LIN {X 0,Y 641.968,Z 762.06,A -85,B 0,C 180,E1 5618.929,E2 5618.929} C_VEL
LIN {X 0,Y 642.524,Z 763.494,A -85,B 0,C 180,E1 5625.268,E2 5625.268} C_VEL
LIN {X 0,Y 669.251,Z 813.676,A -85,B 0,C 180,E1 5628.22,E2 5628.22} C_VEL
LIN {X 0,Y 666.394,Z 892.129,A -85,B 0,C 180,E1 5629.884,E2 5629.884} C_VEL
LIN {X 0,Y 661.27,Z 964.972,A -85,B 0,C 180,E1 5632.787,E2 5632.787} C_VEL
LIN {X 0,Y 655.013,Z 1034.337,A -85,B 0,C 180,E1 5637.06,E2 5637.06} C_VEL
LIN {X 0,Y 649.321,Z 1095.62,A -85,B 0,C 180,E1 5642.548,E2 5642.548} C_VEL
LIN {X 0,Y 645.565,Z 1141.854,A -85,B 0,C 180,E1 5648.388,E2 5648.388} C_VEL
LIN {X 0,Y 643.703,Z 1174.825,A -85,B 0,C 180,E1 5654.309,E2 5654.309} C_VEL
LIN {X 0,Y 643.008,Z 1195.415,A -85,B 0,C 180,E1 5659.842,E2 5659.842} C_VEL
LIN {X 0,Y 642.913,Z 1206.863,A -85,B 0,C 180,E1 5665.298,E2 5665.298} C_VEL
LIN {X 0,Y 643.047,Z 1209.856,A -85,B 0,C 180,E1 5670.712,E2 5670.712} C_VEL
LIN {X 0,Y 642.983,Z 1203.539,A -85,B 0,C 180,E1 5676.768,E2 5676.768} C_VEL
LIN {X 0,Y 643.323,Z 1187.342,A -85,B 0,C 180,E1 5682.645,E2 5682.645} C_VEL
LIN {X 0,Y 644.54,Z 1158.659,A -85,B 0,C 180,E1 5688.859,E2 5688.859} C_VEL
LIN {X 0,Y 647.642,Z 1116.321,A -85,B 0,C 180,E1 5695.063,E2 5695.063} C_VEL
LIN {X 0,Y 652.69,Z 1059.566,A -85,B 0,C 180,E1 5700.912,E2 5700.912} C_VEL
LIN {X 0,Y 658.813,Z 993.276,A -85,B 0,C 180,E1 5705.678,E2 5705.678} C_VEL
LIN {X 0,Y 664.564,Z 922,A -85,B 0,C 180,E1 5709.097,E2 5709.097} C_VEL
LIN {X 0,Y 668.508,Z 847.122,A -85,B 0,C 180,E1 5711.232,E2 5711.232} C_VEL
LIN {X 0,Y 668.062,Z 809.122,A -85,B 0,C 180,E1 5711.936,E2 5711.936} C_VEL
LIN {X 0,Y 645.282,Z 769.291,A -85,B 0,C 180,E1 5714.483,E2 5714.483} C_VEL
LIN {X 0,Y 642.431,Z 762.06,A -85,B 0,C 180,E1 5715.512,E2 5715.512} C_VEL
LIN {X 0,Y 642.499,Z 762.06,A -85,B 0,C 180,E1 5724.625,E2 5724.625} C_VEL
LIN {X 0,Y 642.667,Z 762.06,A -85,B 0,C 180,E1 5732.544,E2 5732.544} C_VEL
LIN {X 0,Y 642.28,Z 762.06,A -85,B 0,C 180,E1 5741.361,E2 5741.361} C_VEL
LIN {X 0,Y 642.684,Z 762.06,A -85,B 0,C 180,E1 5749.761,E2 5749.761} C_VEL
LIN {X 0,Y 643.54,Z 762.06,A -85,B 0,C 180,E1 5759.285,E2 5759.285} C_VEL
LIN {X 0,Y 643.048,Z 762.06,A -85,B 0,C 180,E1 5767.416,E2 5767.416} C_VEL
LIN {X 0,Y 642.573,Z 762.06,A -85,B 0,C 180,E1 5775.715,E2 5775.715} C_VEL
LIN {X 0,Y 642.422,Z 762.06,A -85,B 0,C 180,E1 5784.501,E2 5784.501} C_VEL
LIN {X 0,Y 642.194,Z 762.06,A -85,B 0,C 180,E1 5792.923,E2 5792.923} C_VEL
LIN {X 0,Y 642.123,Z 762.06,A -85,B 0,C 180,E1 5800.473,E2 5800.473} C_VEL
LIN {X 0,Y 642.633,Z 763.835,A -85,B 0,C 180,E1 5805.715,E2 5805.715} C_VEL
LIN {X 0,Y 668.753,Z 814.883,A -85,B 0,C 180,E1 5808.697,E2 5808.697} C_VEL
LIN {X 0,Y 664.877,Z 886.869,A -85,B 0,C 180,E1 5810.661,E2 5810.661} C_VEL
LIN {X 0,Y 659.36,Z 956.9,A -85,B 0,C 180,E1 5813.914,E2 5813.914} C_VEL
LIN {X 0,Y 653.066,Z 1024.664,A -85,B 0,C 180,E1 5818.626,E2 5818.626} C_VEL
LIN {X 0,Y 648.001,Z 1081.384,A -85,B 0,C 180,E1 5824.29,E2 5824.29} C_VEL
LIN {X 0,Y 644.898,Z 1124.533,A -85,B 0,C 180,E1 5830.373,E2 5830.373} C_VEL
LIN {X 0,Y 643.324,Z 1154.863,A -85,B 0,C 180,E1 5836.668,E2 5836.668} C_VEL
LIN {X 0,Y 643.018,Z 1172.142,A -85,B 0,C 180,E1 5842.507,E2 5842.507} C_VEL
LIN {X 0,Y 642.979,Z 1179.378,A -85,B 0,C 180,E1 5847.936,E2 5847.936} C_VEL
LIN {X 0,Y 643.293,Z 1178.365,A -85,B 0,C 180,E1 5853.345,E2 5853.345} C_VEL
LIN {X 0,Y 643.278,Z 1167.177,A -85,B 0,C 180,E1 5859.467,E2 5859.467} C_VEL
LIN {X 0,Y 643.912,Z 1143.027,A -85,B 0,C 180,E1 5866.037,E2 5866.037} C_VEL
LIN {X 0,Y 646.233,Z 1105.047,A -85,B 0,C 180,E1 5872.545,E2 5872.545} C_VEL
LIN {X 0,Y 650.445,Z 1053.564,A -85,B 0,C 180,E1 5878.643,E2 5878.643} C_VEL
LIN {X 0,Y 656.28,Z 990.818,A -85,B 0,C 180,E1 5883.862,E2 5883.862} C_VEL
LIN {X 0,Y 662.363,Z 920.75,A -85,B 0,C 180,E1 5887.851,E2 5887.851} C_VEL
LIN {X 0,Y 667.266,Z 846.885,A -85,B 0,C 180,E1 5890.503,E2 5890.503} C_VEL
LIN {X 0,Y 667.55,Z 807.621,A -85,B 0,C 180,E1 5891.463,E2 5891.463} C_VEL
LIN {X 0,Y 642.29,Z 762.06,A -85,B 0,C 180,E1 5894.401,E2 5894.401} C_VEL
LIN {X 0,Y 642.604,Z 762.06,A -85,B 0,C 180,E1 5903.031,E2 5903.031} C_VEL
LIN {X 0,Y 643.226,Z 764.059,A -85,B 0,C 180,E1 5904.955,E2 5904.955} C_VEL
LIN {X 0,Y 646.792,Z 798.497,A -85,B 0,C 180,E1 5906.449,E2 5906.449} C_VEL
LIN {X 0,Y 645.62,Z 850.108,A -85,B 0,C 180,E1 5908.348,E2 5908.348} C_VEL
LIN {X 0,Y 645.924,Z 977.217,A -85,B 0,C 180,E1 5910.012,E2 5910.012} C_VEL
LIN {X 0,Y 645.226,Z 1016.362,A -85,B 0,C 180,E1 5911.875,E2 5911.875} C_VEL
LIN {X 0,Y 644.386,Z 1044.873,A -85,B 0,C 180,E1 5914.627,E2 5914.627} C_VEL
LIN {X 0,Y 643.963,Z 1061.534,A -85,B 0,C 180,E1 5917.854,E2 5917.854} C_VEL
LIN {X 0,Y 643.934,Z 1066.232,A -85,B 0,C 180,E1 5921.494,E2 5921.494} C_VEL
LIN {X 0,Y 644.339,Z 1057.329,A -85,B 0,C 180,E1 5925.23,E2 5925.23} C_VEL
LIN {X 0,Y 644.899,Z 1035.187,A -85,B 0,C 180,E1 5928.505,E2 5928.505} C_VEL
LIN {X 0,Y 645.628,Z 1002.226,A -85,B 0,C 180,E1 5930.925,E2 5930.925} C_VEL
LIN {X 0,Y 645.974,Z 962.512,A -85,B 0,C 180,E1 5932.236,E2 5932.236} C_VEL
LIN {X 0,Y 646.109,Z 839.86,A -85,B 0,C 180,E1 5933.847,E2 5933.847} C_VEL
LIN {X 0,Y 644.772,Z 767.664,A -85,B 0,C 180,E1 5936.755,E2 5936.755} C_VEL
LIN {X 0,Y 643.716,Z 762.06,A -85,B 0,C 180,E1 5937.013,E2 5937.013} C_VEL
LIN {X 0,Y 642.836,Z 762.06,A -85,B 0,C 180,E1 5946.137,E2 5946.137} C_VEL
LIN {X 0,Y 642.506,Z 762.06,A -85,B 0,C 180,E1 5954.397,E2 5954.397} C_VEL
LIN {X 0,Y 642.148,Z 762.06,A -85,B 0,C 180,E1 5962.989,E2 5962.989} C_VEL
LIN {X 0,Y 642.281,Z 762.06,A -85,B 0,C 180,E1 5970.57,E2 5970.57} C_VEL
LIN {X 0,Y 641.968,Z 762.06,A -85,B 0,C 180,E1 5978.929,E2 5978.929} C_VEL
LIN {X 0,Y 633.847,Z 762.06,A -85,B 0,C 180,E1 5982.023,E2 5982.023} C_VEL
LIN {X 0,Y 634.54,Z 763.771,A -85,B 0,C 180,E1 5984.577,E2 5984.577} C_VEL
LIN {X 0,Y 663.265,Z 815.131,A -85,B 0,C 180,E1 5987.777,E2 5987.777} C_VEL
LIN {X 0,Y 660.138,Z 893.604,A -85,B 0,C 180,E1 5989.476,E2 5989.476} C_VEL
LIN {X 0,Y 654.741,Z 964.946,A -85,B 0,C 180,E1 5992.35,E2 5992.35} C_VEL
LIN {X 0,Y 648.038,Z 1034.342,A -85,B 0,C 180,E1 5996.659,E2 5996.659} C_VEL
LIN {X 0,Y 641.865,Z 1095.691,A -85,B 0,C 180,E1 6002.209,E2 6002.209} C_VEL
LIN {X 0,Y 637.775,Z 1142.428,A -85,B 0,C 180,E1 6008.198,E2 6008.198} C_VEL
LIN {X 0,Y 635.806,Z 1174.828,A -85,B 0,C 180,E1 6014.109,E2 6014.109} C_VEL
LIN {X 0,Y 635.06,Z 1195.414,A -85,B 0,C 180,E1 6019.714,E2 6019.714} C_VEL
LIN {X 0,Y 634.932,Z 1206.862,A -85,B 0,C 180,E1 6025.239,E2 6025.239} C_VEL
LIN {X 0,Y 635.041,Z 1209.858,A -85,B 0,C 180,E1 6030.721,E2 6030.721} C_VEL
LIN {X 0,Y 634.928,Z 1203.138,A -85,B 0,C 180,E1 6037.068,E2 6037.068} C_VEL
LIN {X 0,Y 635.323,Z 1186.051,A -85,B 0,C 180,E1 6043.151,E2 6043.151} C_VEL
LIN {X 0,Y 636.725,Z 1157.895,A -85,B 0,C 180,E1 6049.239,E2 6049.239} C_VEL
LIN {X 0,Y 640.117,Z 1115.788,A -85,B 0,C 180,E1 6055.446,E2 6055.446} C_VEL
LIN {X 0,Y 645.467,Z 1059.914,A -85,B 0,C 180,E1 6061.264,E2 6061.264} C_VEL
LIN {X 0,Y 652.198,Z 992.447,A -85,B 0,C 180,E1 6066.149,E2 6066.149} C_VEL
LIN {X 0,Y 658.226,Z 922.276,A -85,B 0,C 180,E1 6069.535,E2 6069.535} C_VEL
LIN {X 0,Y 662.458,Z 847.779,A -85,B 0,C 180,E1 6071.678,E2 6071.678} C_VEL
LIN {X 0,Y 662.128,Z 812.528,A -85,B 0,C 180,E1 6072.35,E2 6072.35} C_VEL
LIN {X 0,Y 634.409,Z 762.06,A -85,B 0,C 180,E1 6075.739,E2 6075.739} C_VEL
LIN {X 0,Y 634.427,Z 762.06,A -85,B 0,C 180,E1 6084.082,E2 6084.082} C_VEL
LIN {X 0,Y 634.647,Z 762.06,A -85,B 0,C 180,E1 6092.168,E2 6092.168} C_VEL
LIN {X 0,Y 634.098,Z 762.06,A -85,B 0,C 180,E1 6099.656,E2 6099.656} C_VEL
LIN {X 0,Y 634.253,Z 762.06,A -85,B 0,C 180,E1 6106.823,E2 6106.823} C_VEL
LIN {X 0,Y 634.501,Z 762.06,A -85,B 0,C 180,E1 6113.782,E2 6113.782} C_VEL
LIN {X 0,Y 634.818,Z 762.06,A -85,B 0,C 180,E1 6120.645,E2 6120.645} C_VEL
LIN {X 0,Y 634.505,Z 762.06,A -85,B 0,C 180,E1 6128.901,E2 6128.901} C_VEL
LIN {X 0,Y 634.515,Z 762.06,A -85,B 0,C 180,E1 6135.919,E2 6135.919} C_VEL
LIN {X 0,Y 634.395,Z 762.06,A -85,B 0,C 180,E1 6144.698,E2 6144.698} C_VEL
LIN {X 0,Y 634.212,Z 762.06,A -85,B 0,C 180,E1 6152.519,E2 6152.519} C_VEL
LIN {X 0,Y 634.111,Z 762.06,A -85,B 0,C 180,E1 6161.094,E2 6161.094} C_VEL
LIN {X 0,Y 634.666,Z 763.885,A -85,B 0,C 180,E1 6165.106,E2 6165.106} C_VEL
LIN {X 0,Y 662.682,Z 816.434,A -85,B 0,C 180,E1 6168.27,E2 6168.27} C_VEL
LIN {X 0,Y 658.534,Z 887.804,A -85,B 0,C 180,E1 6170.246,E2 6170.246} C_VEL
LIN {X 0,Y 652.535,Z 958.678,A -85,B 0,C 180,E1 6173.589,E2 6173.589} C_VEL
LIN {X 0,Y 645.795,Z 1026.081,A -85,B 0,C 180,E1 6178.361,E2 6178.361} C_VEL
LIN {X 0,Y 640.299,Z 1083.145,A -85,B 0,C 180,E1 6184.18,E2 6184.18} C_VEL
LIN {X 0,Y 637.011,Z 1125.632,A -85,B 0,C 180,E1 6190.321,E2 6190.321} C_VEL
LIN {X 0,Y 635.418,Z 1154.859,A -85,B 0,C 180,E1 6196.499,E2 6196.499} C_VEL
LIN {X 0,Y 635.052,Z 1172.138,A -85,B 0,C 180,E1 6202.412,E2 6202.412} C_VEL
LIN {X 0,Y 634.984,Z 1179.375,A -85,B 0,C 180,E1 6207.91,E2 6207.91} C_VEL
LIN {X 0,Y 635.269,Z 1178.363,A -85,B 0,C 180,E1 6213.387,E2 6213.387} C_VEL
LIN {X 0,Y 635.253,Z 1167.176,A -85,B 0,C 180,E1 6219.588,E2 6219.588} C_VEL
LIN {X 0,Y 635.98,Z 1143.03,A -85,B 0,C 180,E1 6226.242,E2 6226.242} C_VEL
LIN {X 0,Y 638.426,Z 1106.075,A -85,B 0,C 180,E1 6232.682,E2 6232.682} C_VEL
LIN {X 0,Y 642.88,Z 1056.271,A -85,B 0,C 180,E1 6238.725,E2 6238.725} C_VEL
LIN {X 0,Y 649.115,Z 993.86,A -85,B 0,C 180,E1 6244.057,E2 6244.057} C_VEL
LIN {X 0,Y 655.63,Z 924.375,A -85,B 0,C 180,E1 6248.126,E2 6248.126} C_VEL
LIN {X 0,Y 660.958,Z 849.366,A -85,B 0,C 180,E1 6250.895,E2 6250.895} C_VEL
LIN {X 0,Y 661.473,Z 810.895,A -85,B 0,C 180,E1 6251.859,E2 6251.859} C_VEL
LIN {X 0,Y 634.183,Z 762.06,A -85,B 0,C 180,E1 6254.984,E2 6254.984} C_VEL
LIN {X 0,Y 634.775,Z 762.06,A -85,B 0,C 180,E1 6264.204,E2 6264.204} C_VEL
LIN {X 0,Y 635.208,Z 764.323,A -85,B 0,C 180,E1 6264.759,E2 6264.759} C_VEL
LIN {X 0,Y 639.068,Z 798.715,A -85,B 0,C 180,E1 6266.267,E2 6266.267} C_VEL
LIN {X 0,Y 637.85,Z 852.278,A -85,B 0,C 180,E1 6268.22,E2 6268.22} C_VEL
LIN {X 0,Y 638.083,Z 977.294,A -85,B 0,C 180,E1 6269.869,E2 6269.869} C_VEL
LIN {X 0,Y 637.407,Z 1016.556,A -85,B 0,C 180,E1 6271.722,E2 6271.722} C_VEL
LIN {X 0,Y 636.506,Z 1046.311,A -85,B 0,C 180,E1 6274.612,E2 6274.612} C_VEL
LIN {X 0,Y 636.047,Z 1064.021,A -85,B 0,C 180,E1 6278.343,E2 6278.343} C_VEL
LIN {X 0,Y 636.029,Z 1067.446,A -85,B 0,C 180,E1 6281.256,E2 6281.256} C_VEL
LIN {X 0,Y 636.402,Z 1058.845,A -85,B 0,C 180,E1 6285.192,E2 6285.192} C_VEL
LIN {X 0,Y 637.035,Z 1036.809,A -85,B 0,C 180,E1 6288.535,E2 6288.535} C_VEL
LIN {X 0,Y 637.827,Z 1002.479,A -85,B 0,C 180,E1 6291.078,E2 6291.078} C_VEL
LIN {X 0,Y 638.126,Z 961.21,A -85,B 0,C 180,E1 6292.397,E2 6292.397} C_VEL
LIN {X 0,Y 638.365,Z 840.977,A -85,B 0,C 180,E1 6293.986,E2 6293.986} C_VEL
LIN {X 0,Y 637.097,Z 769.419,A -85,B 0,C 180,E1 6296.883,E2 6296.883} C_VEL
LIN {X 0,Y 635.567,Z 762.06,A -85,B 0,C 180,E1 6297.304,E2 6297.304} C_VEL
LIN {X 0,Y 634.794,Z 762.06,A -85,B 0,C 180,E1 6306.215,E2 6306.215} C_VEL
LIN {X 0,Y 634.463,Z 762.06,A -85,B 0,C 180,E1 6314.584,E2 6314.584} C_VEL
LIN {X 0,Y 634.161,Z 762.06,A -85,B 0,C 180,E1 6322.995,E2 6322.995} C_VEL
LIN {X 0,Y 634.168,Z 762.06,A -85,B 0,C 180,E1 6331.003,E2 6331.003} C_VEL
LIN {X 0,Y 633.915,Z 762.06,A -85,B 0,C 180,E1 6339.418,E2 6339.418} C_VEL
LIN {X 0,Y 633.847,Z 762.06,A -85,B 0,C 180,E1 6342.023,E2 6342.023} C_VEL
LIN {X 0,Y 626.067,Z 762.06,A -85,B 0,C 180,E1 6343.324,E2 6343.324} C_VEL
LIN {X 0,Y 626.693,Z 764.76,A -85,B 0,C 180,E1 6343.865,E2 6343.865} C_VEL
LIN {X 0,Y 657.298,Z 819.468,A -85,B 0,C 180,E1 6347.369,E2 6347.369} C_VEL
LIN {X 0,Y 653.635,Z 898.642,A -85,B 0,C 180,E1 6349.17,E2 6349.17} C_VEL
LIN {X 0,Y 647.505,Z 972.54,A -85,B 0,C 180,E1 6352.296,E2 6352.296} C_VEL
LIN {X 0,Y 640.367,Z 1040.903,A -85,B 0,C 180,E1 6356.759,E2 6356.759} C_VEL
LIN {X 0,Y 634.008,Z 1100.059,A -85,B 0,C 180,E1 6362.346,E2 6362.346} C_VEL
LIN {X 0,Y 629.741,Z 1147.139,A -85,B 0,C 180,E1 6368.671,E2 6368.671} C_VEL
LIN {X 0,Y 627.746,Z 1180.061,A -85,B 0,C 180,E1 6375.127,E2 6375.127} C_VEL
LIN {X 0,Y 627.122,Z 1200.734,A -85,B 0,C 180,E1 6381.69,E2 6381.69} C_VEL
LIN {X 0,Y 627.224,Z 1209.409,A -85,B 0,C 180,E1 6387.957,E2 6387.957} C_VEL
LIN {X 0,Y 627.441,Z 1206.762,A -85,B 0,C 180,E1 6394.892,E2 6394.892} C_VEL
LIN {X 0,Y 627.557,Z 1190.935,A -85,B 0,C 180,E1 6401.897,E2 6401.897} C_VEL
LIN {X 0,Y 628.717,Z 1162.227,A -85,B 0,C 180,E1 6408.688,E2 6408.688} C_VEL
LIN {X 0,Y 632.127,Z 1121.002,A -85,B 0,C 180,E1 6415.117,E2 6415.117} C_VEL
LIN {X 0,Y 637.853,Z 1064.411,A -85,B 0,C 180,E1 6421.25,E2 6421.25} C_VEL
LIN {X 0,Y 644.857,Z 998.953,A -85,B 0,C 180,E1 6426.185,E2 6426.185} C_VEL
LIN {X 0,Y 651.596,Z 927.003,A -85,B 0,C 180,E1 6429.808,E2 6429.808} C_VEL
LIN {X 0,Y 656.296,Z 851.279,A -85,B 0,C 180,E1 6432.08,E2 6432.08} C_VEL
LIN {X 0,Y 656.226,Z 815.81,A -85,B 0,C 180,E1 6432.773,E2 6432.773} C_VEL
LIN {X 0,Y 626.346,Z 762.06,A -85,B 0,C 180,E1 6436.284,E2 6436.284} C_VEL
LIN {X 0,Y 626.397,Z 762.06,A -85,B 0,C 180,E1 6445.255,E2 6445.255} C_VEL
LIN {X 0,Y 626.646,Z 762.06,A -85,B 0,C 180,E1 6453.344,E2 6453.344} C_VEL
LIN {X 0,Y 626.588,Z 762.06,A -85,B 0,C 180,E1 6463.17,E2 6463.17} C_VEL
LIN {X 0,Y 626.933,Z 762.06,A -85,B 0,C 180,E1 6472.31,E2 6472.31} C_VEL
LIN {X 0,Y 626.825,Z 762.06,A -85,B 0,C 180,E1 6480.653,E2 6480.653} C_VEL
LIN {X 0,Y 626.47,Z 762.06,A -85,B 0,C 180,E1 6489.016,E2 6489.016} C_VEL
LIN {X 0,Y 626.268,Z 762.06,A -85,B 0,C 180,E1 6496.733,E2 6496.733} C_VEL
LIN {X 0,Y 626.356,Z 762.06,A -85,B 0,C 180,E1 6505.037,E2 6505.037} C_VEL
LIN {X 0,Y 626.128,Z 762.06,A -85,B 0,C 180,E1 6513.206,E2 6513.206} C_VEL
LIN {X 0,Y 626.073,Z 762.06,A -85,B 0,C 180,E1 6521.739,E2 6521.739} C_VEL
LIN {X 0,Y 626.592,Z 764.01,A -85,B 0,C 180,E1 6524.571,E2 6524.571} C_VEL
LIN {X 0,Y 656.59,Z 819.093,A -85,B 0,C 180,E1 6527.857,E2 6527.857} C_VEL
LIN {X 0,Y 652.184,Z 888.957,A -85,B 0,C 180,E1 6529.833,E2 6529.833} C_VEL
LIN {X 0,Y 645.737,Z 960.133,A -85,B 0,C 180,E1 6533.237,E2 6533.237} C_VEL
LIN {X 0,Y 638.566,Z 1027.116,A -85,B 0,C 180,E1 6538.056,E2 6538.056} C_VEL
LIN {X 0,Y 632.662,Z 1084.177,A -85,B 0,C 180,E1 6543.978,E2 6543.978} C_VEL
LIN {X 0,Y 629.016,Z 1127.554,A -85,B 0,C 180,E1 6550.417,E2 6550.417} C_VEL
LIN {X 0,Y 627.372,Z 1156.195,A -85,B 0,C 180,E1 6556.679,E2 6556.679} C_VEL
LIN {X 0,Y 626.932,Z 1173.543,A -85,B 0,C 180,E1 6563.012,E2 6563.012} C_VEL
LIN {X 0,Y 627.016,Z 1179.371,A -85,B 0,C 180,E1 6567.883,E2 6567.883} C_VEL
LIN {X 0,Y 627.263,Z 1178.361,A -85,B 0,C 180,E1 6573.43,E2 6573.43} C_VEL
LIN {X 0,Y 627.229,Z 1167.174,A -85,B 0,C 180,E1 6579.712,E2 6579.712} C_VEL
LIN {X 0,Y 628.05,Z 1143.033,A -85,B 0,C 180,E1 6586.453,E2 6586.453} C_VEL
LIN {X 0,Y 630.652,Z 1106.779,A -85,B 0,C 180,E1 6592.871,E2 6592.871} C_VEL
LIN {X 0,Y 635.435,Z 1056.483,A -85,B 0,C 180,E1 6599.071,E2 6599.071} C_VEL
LIN {X 0,Y 642.265,Z 993.446,A -85,B 0,C 180,E1 6604.503,E2 6604.503} C_VEL
LIN {X 0,Y 649.286,Z 923.399,A -85,B 0,C 180,E1 6608.617,E2 6608.617} C_VEL
LIN {X 0,Y 654.948,Z 849.132,A -85,B 0,C 180,E1 6611.36,E2 6611.36} C_VEL
LIN {X 0,Y 655.201,Z 813.703,A -85,B 0,C 180,E1 6612.287,E2 6612.287} C_VEL
LIN {X 0,Y 626.1,Z 762.06,A -85,B 0,C 180,E1 6615.584,E2 6615.584} C_VEL
LIN {X 0,Y 626.856,Z 762.599,A -85,B 0,C 180,E1 6624.465,E2 6624.465} C_VEL
LIN {X 0,Y 631.343,Z 799.212,A -85,B 0,C 180,E1 6626.092,E2 6626.092} C_VEL
LIN {X 0,Y 630.035,Z 850.807,A -85,B 0,C 180,E1 6628.044,E2 6628.044} C_VEL
LIN {X 0,Y 630.259,Z 978.804,A -85,B 0,C 180,E1 6629.761,E2 6629.761} C_VEL
LIN {X 0,Y 629.552,Z 1017.575,A -85,B 0,C 180,E1 6631.621,E2 6631.621} C_VEL
LIN {X 0,Y 628.63,Z 1047.399,A -85,B 0,C 180,E1 6634.548,E2 6634.548} C_VEL
LIN {X 0,Y 628.128,Z 1065.171,A -85,B 0,C 180,E1 6638.339,E2 6638.339} C_VEL
LIN {X 0,Y 628.143,Z 1067.58,A -85,B 0,C 180,E1 6642.469,E2 6642.469} C_VEL
LIN {X 0,Y 628.805,Z 1054.986,A -85,B 0,C 180,E1 6646.257,E2 6646.257} C_VEL
LIN {X 0,Y 629.202,Z 1029.368,A -85,B 0,C 180,E1 6649.446,E2 6649.446} C_VEL
LIN {X 0,Y 630.045,Z 992.652,A -85,B 0,C 180,E1 6651.69,E2 6651.69} C_VEL
LIN {X 0,Y 630.237,Z 948.788,A -85,B 0,C 180,E1 6652.693,E2 6652.693} C_VEL
LIN {X 0,Y 630.616,Z 842.225,A -85,B 0,C 180,E1 6654.128,E2 6654.128} C_VEL
LIN {X 0,Y 629.127,Z 769.513,A -85,B 0,C 180,E1 6657.086,E2 6657.086} C_VEL
LIN {X 0,Y 627.391,Z 762.06,A -85,B 0,C 180,E1 6657.615,E2 6657.615} C_VEL
LIN {X 0,Y 626.764,Z 762.06,A -85,B 0,C 180,E1 6666.295,E2 6666.295} C_VEL
LIN {X 0,Y 626.397,Z 762.06,A -85,B 0,C 180,E1 6674.776,E2 6674.776} C_VEL
LIN {X 0,Y 626.304,Z 762.06,A -85,B 0,C 180,E1 6682.099,E2 6682.099} C_VEL
LIN {X 0,Y 626.176,Z 762.06,A -85,B 0,C 180,E1 6690.73,E2 6690.73} C_VEL
LIN {X 0,Y 626.052,Z 762.06,A -85,B 0,C 180,E1 6698.222,E2 6698.222} C_VEL
LIN {X 0,Y 626.067,Z 762.06,A -85,B 0,C 180,E1 6703.324,E2 6703.324} C_VEL
LIN {X 0,Y 629.491,Z 771.34,A -85,B 0,C 180,E1 6704.231,E2 6704.231} C_VEL
LIN {X 0,Y 634.953,Z 790.895,A -85,B 0,C 180,E1 6705.038,E2 6705.038} C_VEL
LIN {X 0,Y 651.282,Z 823.776,A -85,B 0,C 180,E1 6706.953,E2 6706.953} C_VEL
LIN {X 0,Y 647.186,Z 902.445,A -85,B 0,C 180,E1 6708.826,E2 6708.826} C_VEL
LIN {X 0,Y 640.779,Z 974.627,A -85,B 0,C 180,E1 6711.959,E2 6711.959} C_VEL
LIN {X 0,Y 633.183,Z 1042.781,A -85,B 0,C 180,E1 6716.494,E2 6716.494} C_VEL
LIN {X 0,Y 626.377,Z 1102.132,A -85,B 0,C 180,E1 6722.231,E2 6722.231} C_VEL
LIN {X 0,Y 621.875,Z 1148.587,A -85,B 0,C 180,E1 6728.633,E2 6728.633} C_VEL
LIN {X 0,Y 619.788,Z 1180.913,A -85,B 0,C 180,E1 6735.143,E2 6735.143} C_VEL
LIN {X 0,Y 619.103,Z 1200.733,A -85,B 0,C 180,E1 6741.582,E2 6741.582} C_VEL
LIN {X 0,Y 619.209,Z 1209.407,A -85,B 0,C 180,E1 6747.931,E2 6747.931} C_VEL
LIN {X 0,Y 619.424,Z 1206.76,A -85,B 0,C 180,E1 6754.956,E2 6754.956} C_VEL
LIN {X 0,Y 619.521,Z 1190.933,A -85,B 0,C 180,E1 6762.054,E2 6762.054} C_VEL
LIN {X 0,Y 620.835,Z 1162.227,A -85,B 0,C 180,E1 6768.934,E2 6768.934} C_VEL
LIN {X 0,Y 624.534,Z 1121.232,A -85,B 0,C 180,E1 6775.412,E2 6775.412} C_VEL
LIN {X 0,Y 630.62,Z 1064.926,A -85,B 0,C 180,E1 6781.599,E2 6781.599} C_VEL
LIN {X 0,Y 638.103,Z 999.563,A -85,B 0,C 180,E1 6786.586,E2 6786.586} C_VEL
LIN {X 0,Y 645.307,Z 927.429,A -85,B 0,C 180,E1 6790.256,E2 6790.256} C_VEL
LIN {X 0,Y 650.302,Z 852.125,A -85,B 0,C 180,E1 6792.538,E2 6792.538} C_VEL
LIN {X 0,Y 650.083,Z 818.594,A -85,B 0,C 180,E1 6793.233,E2 6793.233} C_VEL
LIN {X 0,Y 618.191,Z 762.06,A -85,B 0,C 180,E1 6797.039,E2 6797.039} C_VEL
LIN {X 0,Y 618.423,Z 762.06,A -85,B 0,C 180,E1 6806.445,E2 6806.445} C_VEL
LIN {X 0,Y 618.654,Z 762.06,A -85,B 0,C 180,E1 6814.538,E2 6814.538} C_VEL
LIN {X 0,Y 618.621,Z 762.06,A -85,B 0,C 180,E1 6823.574,E2 6823.574} C_VEL
LIN {X 0,Y 618.937,Z 762.06,A -85,B 0,C 180,E1 6832.21,E2 6832.21} C_VEL
LIN {X 0,Y 618.818,Z 762.06,A -85,B 0,C 180,E1 6840.661,E2 6840.661} C_VEL
LIN {X 0,Y 618.918,Z 762.06,A -85,B 0,C 180,E1 6847.707,E2 6847.707} C_VEL
LIN {X 0,Y 618.368,Z 762.06,A -85,B 0,C 180,E1 6856.347,E2 6856.347} C_VEL
LIN {X 0,Y 618.297,Z 762.06,A -85,B 0,C 180,E1 6865.386,E2 6865.386} C_VEL
LIN {X 0,Y 618.116,Z 762.06,A -85,B 0,C 180,E1 6873.475,E2 6873.475} C_VEL
LIN {X 0,Y 618.107,Z 762.06,A -85,B 0,C 180,E1 6882.401,E2 6882.401} C_VEL
LIN {X 0,Y 618.351,Z 763.179,A -85,B 0,C 180,E1 6884.005,E2 6884.005} C_VEL
LIN {X 0,Y 646.298,Z 813.112,A -85,B 0,C 180,E1 6886.887,E2 6886.887} C_VEL
LIN {X 0,Y 650.316,Z 825.734,A -85,B 0,C 180,E1 6887.511,E2 6887.511} C_VEL
LIN {X 0,Y 645.298,Z 896.483,A -85,B 0,C 180,E1 6889.665,E2 6889.665} C_VEL
LIN {X 0,Y 638.396,Z 966.596,A -85,B 0,C 180,E1 6893.181,E2 6893.181} C_VEL
LIN {X 0,Y 630.748,Z 1033.572,A -85,B 0,C 180,E1 6898.227,E2 6898.227} C_VEL
LIN {X 0,Y 624.631,Z 1089.212,A -85,B 0,C 180,E1 6904.275,E2 6904.275} C_VEL
LIN {X 0,Y 620.913,Z 1130.466,A -85,B 0,C 180,E1 6910.698,E2 6910.698} C_VEL
LIN {X 0,Y 619.325,Z 1157.522,A -85,B 0,C 180,E1 6916.863,E2 6916.863} C_VEL
LIN {X 0,Y 619.016,Z 1173.191,A -85,B 0,C 180,E1 6922.731,E2 6922.731} C_VEL
LIN {X 0,Y 619.02,Z 1179.368,A -85,B 0,C 180,E1 6927.856,E2 6927.856} C_VEL
LIN {X 0,Y 619.241,Z 1178.358,A -85,B 0,C 180,E1 6933.475,E2 6933.475} C_VEL
LIN {X 0,Y 619.22,Z 1167.172,A -85,B 0,C 180,E1 6939.839,E2 6939.839} C_VEL
LIN {X 0,Y 620.106,Z 1144.594,A -85,B 0,C 180,E1 6946.305,E2 6946.305} C_VEL
LIN {X 0,Y 622.842,Z 1108.558,A -85,B 0,C 180,E1 6952.901,E2 6952.901} C_VEL
LIN {X 0,Y 627.926,Z 1058.302,A -85,B 0,C 180,E1 6959.254,E2 6959.254} C_VEL
LIN {X 0,Y 635.176,Z 995.766,A -85,B 0,C 180,E1 6964.762,E2 6964.762} C_VEL
LIN {X 0,Y 642.656,Z 926.328,A -85,B 0,C 180,E1 6968.937,E2 6968.937} C_VEL
LIN {X 0,Y 648.645,Z 851.713,A -85,B 0,C 180,E1 6971.764,E2 6971.764} C_VEL
LIN {X 0,Y 649.372,Z 817.542,A -85,B 0,C 180,E1 6972.667,E2 6972.667} C_VEL
LIN {X 0,Y 622.158,Z 771.6,A -85,B 0,C 180,E1 6975.529,E2 6975.529} C_VEL
LIN {X 0,Y 618.101,Z 762.06,A -85,B 0,C 180,E1 6976.031,E2 6976.031} C_VEL
LIN {X 0,Y 618.986,Z 763.724,A -85,B 0,C 180,E1 6984.288,E2 6984.288} C_VEL
LIN {X 0,Y 623.63,Z 798.932,A -85,B 0,C 180,E1 6985.881,E2 6985.881} C_VEL
LIN {X 0,Y 622.278,Z 855.046,A -85,B 0,C 180,E1 6987.936,E2 6987.936} C_VEL
LIN {X 0,Y 622.431,Z 978.876,A -85,B 0,C 180,E1 6989.611,E2 6989.611} C_VEL
LIN {X 0,Y 621.707,Z 1018.458,A -85,B 0,C 180,E1 6991.507,E2 6991.507} C_VEL
LIN {X 0,Y 620.752,Z 1047.975,A -85,B 0,C 180,E1 6994.411,E2 6994.411} C_VEL
LIN {X 0,Y 620.223,Z 1065.819,A -85,B 0,C 180,E1 6998.14,E2 6998.14} C_VEL
LIN {X 0,Y 620.221,Z 1069.028,A -85,B 0,C 180,E1 7002.238,E2 7002.238} C_VEL
LIN {X 0,Y 620.808,Z 1058.342,A -85,B 0,C 180,E1 7005.896,E2 7005.896} C_VEL
LIN {X 0,Y 621.261,Z 1034.781,A -85,B 0,C 180,E1 7009.132,E2 7009.132} C_VEL
LIN {X 0,Y 622.175,Z 999.631,A -85,B 0,C 180,E1 7011.54,E2 7011.54} C_VEL
LIN {X 0,Y 622.411,Z 957.301,A -85,B 0,C 180,E1 7012.732,E2 7012.732} C_VEL
LIN {X 0,Y 622.859,Z 843.255,A -85,B 0,C 180,E1 7014.274,E2 7014.274} C_VEL
LIN {X 0,Y 621.314,Z 770.745,A -85,B 0,C 180,E1 7017.242,E2 7017.242} C_VEL
LIN {X 0,Y 619.33,Z 762.06,A -85,B 0,C 180,E1 7017.76,E2 7017.76} C_VEL
LIN {X 0,Y 618.575,Z 762.06,A -85,B 0,C 180,E1 7026.883,E2 7026.883} C_VEL
LIN {X 0,Y 618.358,Z 762.06,A -85,B 0,C 180,E1 7034.973,E2 7034.973} C_VEL
LIN {X 0,Y 618.104,Z 762.06,A -85,B 0,C 180,E1 7043.088,E2 7043.088} C_VEL
LIN {X 0,Y 618.008,Z 762.06,A -85,B 0,C 180,E1 7051.908,E2 7051.908} C_VEL
LIN {X 0,Y 617.796,Z 762.06,A -85,B 0,C 180,E1 7060.657,E2 7060.657} C_VEL
LIN {X 0,Y 618.198,Z 763.848,A -85,B 0,C 180,E1 7063.029,E2 7063.029} C_VEL
LIN {X 0,Y 634.953,Z 790.895,A -85,B 0,C 180,E1 7065.038,E2 7065.038} C_VEL
LIN {X 0,Y 644.233,Z 822.02,A -85,B 0,C 180,E1 7066.332,E2 7066.332} C_VEL
LIN {X 0,Y 641.041,Z 903.216,A -85,B 0,C 180,E1 7068.375,E2 7068.375} C_VEL
LIN {X 0,Y 634.108,Z 976.405,A -85,B 0,C 180,E1 7071.598,E2 7071.598} C_VEL
LIN {X 0,Y 626.061,Z 1044.137,A -85,B 0,C 180,E1 7076.18,E2 7076.18} C_VEL
LIN {X 0,Y 618.721,Z 1104.378,A -85,B 0,C 180,E1 7082.136,E2 7082.136} C_VEL
LIN {X 0,Y 613.996,Z 1151.061,A -85,B 0,C 180,E1 7088.771,E2 7088.771} C_VEL
LIN {X 0,Y 611.931,Z 1184.327,A -85,B 0,C 180,E1 7095.861,E2 7095.861} C_VEL
LIN {X 0,Y 611.493,Z 1203.622,A -85,B 0,C 180,E1 7102.926,E2 7102.926} C_VEL
LIN {X 0,Y 611.631,Z 1209.878,A -85,B 0,C 180,E1 7109.327,E2 7109.327} C_VEL
LIN {X 0,Y 611.081,Z 1204.687,A -85,B 0,C 180,E1 7116.453,E2 7116.453} C_VEL
LIN {X 0,Y 611.424,Z 1188.58,A -85,B 0,C 180,E1 7122.944,E2 7122.944} C_VEL
LIN {X 0,Y 612.986,Z 1162.226,A -85,B 0,C 180,E1 7129.186,E2 7129.186} C_VEL
LIN {X 0,Y 617.012,Z 1120.689,A -85,B 0,C 180,E1 7135.821,E2 7135.821} C_VEL
LIN {X 0,Y 623.439,Z 1065.251,A -85,B 0,C 180,E1 7141.972,E2 7141.972} C_VEL
LIN {X 0,Y 631.438,Z 999.664,A -85,B 0,C 180,E1 7147.029,E2 7147.029} C_VEL
LIN {X 0,Y 638.954,Z 929.065,A -85,B 0,C 180,E1 7150.661,E2 7150.661} C_VEL
LIN {X 0,Y 644.343,Z 853.012,A -85,B 0,C 180,E1 7153.003,E2 7153.003} C_VEL
LIN {X 0,Y 644.265,Z 822.055,A -85,B 0,C 180,E1 7153.665,E2 7153.665} C_VEL
LIN {X 0,Y 610.086,Z 762.06,A -85,B 0,C 180,E1 7157.875,E2 7157.875} C_VEL
LIN {X 0,Y 610.429,Z 762.06,A -85,B 0,C 180,E1 7166.446,E2 7166.446} C_VEL
LIN {X 0,Y 610.566,Z 762.06,A -85,B 0,C 180,E1 7175.194,E2 7175.194} C_VEL
LIN {X 0,Y 610.518,Z 762.06,A -85,B 0,C 180,E1 7184.831,E2 7184.831} C_VEL
LIN {X 0,Y 610.557,Z 762.06,A -85,B 0,C 180,E1 7193.537,E2 7193.537} C_VEL
LIN {X 0,Y 610.811,Z 762.06,A -85,B 0,C 180,E1 7200.67,E2 7200.67} C_VEL
LIN {X 0,Y 610.865,Z 762.06,A -85,B 0,C 180,E1 7207.809,E2 7207.809} C_VEL
LIN {X 0,Y 610.266,Z 762.06,A -85,B 0,C 180,E1 7216.684,E2 7216.684} C_VEL
LIN {X 0,Y 610.311,Z 762.06,A -85,B 0,C 180,E1 7224.754,E2 7224.754} C_VEL
LIN {X 0,Y 610.138,Z 762.06,A -85,B 0,C 180,E1 7233.513,E2 7233.513} C_VEL
LIN {X 0,Y 610.114,Z 762.06,A -85,B 0,C 180,E1 7242.751,E2 7242.751} C_VEL
LIN {X 0,Y 610.417,Z 763.805,A -85,B 0,C 180,E1 7243.471,E2 7243.471} C_VEL
LIN {X 0,Y 641.715,Z 819.226,A -85,B 0,C 180,E1 7246.65,E2 7246.65} C_VEL
LIN {X 0,Y 644.054,Z 831.064,A -85,B 0,C 180,E1 7247.148,E2 7247.148} C_VEL
LIN {X 0,Y 638.7,Z 901.199,A -85,B 0,C 180,E1 7249.386,E2 7249.386} C_VEL
LIN {X 0,Y 631.239,Z 971.064,A -85,B 0,C 180,E1 7253.018,E2 7253.018} C_VEL
LIN {X 0,Y 623.239,Z 1036.755,A -85,B 0,C 180,E1 7258.122,E2 7258.122} C_VEL
LIN {X 0,Y 616.79,Z 1091.621,A -85,B 0,C 180,E1 7264.261,E2 7264.261} C_VEL
LIN {X 0,Y 613.135,Z 1130.462,A -85,B 0,C 180,E1 7270.443,E2 7270.443} C_VEL
LIN {X 0,Y 611.329,Z 1158.73,A -85,B 0,C 180,E1 7277.054,E2 7277.054} C_VEL
LIN {X 0,Y 611.038,Z 1173.19,A -85,B 0,C 180,E1 7282.636,E2 7282.636} C_VEL
LIN {X 0,Y 611.024,Z 1179.364,A -85,B 0,C 180,E1 7287.828,E2 7287.828} C_VEL
LIN {X 0,Y 611.221,Z 1178.356,A -85,B 0,C 180,E1 7293.52,E2 7293.52} C_VEL
LIN {X 0,Y 611.195,Z 1167.171,A -85,B 0,C 180,E1 7299.969,E2 7299.969} C_VEL
LIN {X 0,Y 612.165,Z 1144.597,A -85,B 0,C 180,E1 7306.522,E2 7306.522} C_VEL
LIN {X 0,Y 615.031,Z 1109.786,A -85,B 0,C 180,E1 7313.016,E2 7313.016} C_VEL
LIN {X 0,Y 620.518,Z 1059.047,A -85,B 0,C 180,E1 7319.555,E2 7319.555} C_VEL
LIN {X 0,Y 628.249,Z 996.316,A -85,B 0,C 180,E1 7325.158,E2 7325.158} C_VEL
LIN {X 0,Y 636.198,Z 927.016,A -85,B 0,C 180,E1 7329.371,E2 7329.371} C_VEL
LIN {X 0,Y 642.557,Z 852.954,A -85,B 0,C 180,E1 7332.206,E2 7332.206} C_VEL
LIN {X 0,Y 643.062,Z 820.145,A -85,B 0,C 180,E1 7333.125,E2 7333.125} C_VEL
LIN {X 0,Y 615.008,Z 773.214,A -85,B 0,C 180,E1 7335.987,E2 7335.987} C_VEL
LIN {X 0,Y 610.091,Z 762.06,A -85,B 0,C 180,E1 7336.59,E2 7336.59} C_VEL
LIN {X 0,Y 610.977,Z 763.863,A -85,B 0,C 180,E1 7344.072,E2 7344.072} C_VEL
LIN {X 0,Y 615.88,Z 800.826,A -85,B 0,C 180,E1 7345.752,E2 7345.752} C_VEL
LIN {X 0,Y 614.493,Z 855.321,A -85,B 0,C 180,E1 7347.774,E2 7347.774} C_VEL
LIN {X 0,Y 614.608,Z 980.528,A -85,B 0,C 180,E1 7349.501,E2 7349.501} C_VEL
LIN {X 0,Y 613.852,Z 1018.741,A -85,B 0,C 180,E1 7351.35,E2 7351.35} C_VEL
LIN {X 0,Y 612.858,Z 1049.261,A -85,B 0,C 180,E1 7354.372,E2 7354.372} C_VEL
LIN {X 0,Y 612.319,Z 1067.168,A -85,B 0,C 180,E1 7358.217,E2 7358.217} C_VEL
LIN {X 0,Y 612.33,Z 1070.447,A -85,B 0,C 180,E1 7362.001,E2 7362.001} C_VEL
LIN {X 0,Y 612.855,Z 1060.543,A -85,B 0,C 180,E1 7365.709,E2 7365.709} C_VEL
LIN {X 0,Y 613.41,Z 1036.402,A -85,B 0,C 180,E1 7369.171,E2 7369.171} C_VEL
LIN {X 0,Y 614.346,Z 1002.249,A -85,B 0,C 180,E1 7371.584,E2 7371.584} C_VEL
LIN {X 0,Y 614.613,Z 961.595,A -85,B 0,C 180,E1 7372.818,E2 7372.818} C_VEL
LIN {X 0,Y 615.115,Z 844.501,A -85,B 0,C 180,E1 7374.424,E2 7374.424} C_VEL
LIN {X 0,Y 613.634,Z 772.497,A -85,B 0,C 180,E1 7377.384,E2 7377.384} C_VEL
LIN {X 0,Y 611.256,Z 762.06,A -85,B 0,C 180,E1 7377.908,E2 7377.908} C_VEL
LIN {X 0,Y 610.698,Z 762.06,A -85,B 0,C 180,E1 7386.461,E2 7386.461} C_VEL
LIN {X 0,Y 610.302,Z 762.06,A -85,B 0,C 180,E1 7395.175,E2 7395.175} C_VEL
LIN {X 0,Y 610.176,Z 762.06,A -85,B 0,C 180,E1 7402.715,E2 7402.715} C_VEL
LIN {X 0,Y 610.095,Z 762.06,A -85,B 0,C 180,E1 7410.977,E2 7410.977} C_VEL
LIN {X 0,Y 609.86,Z 762.06,A -85,B 0,C 180,E1 7419.43,E2 7419.43} C_VEL
LIN {X 0,Y 610.161,Z 764.094,A -85,B 0,C 180,E1 7422.223,E2 7422.223} C_VEL
LIN {X 0,Y 644.233,Z 822.02,A -85,B 0,C 180,E1 7426.332,E2 7426.332} C_VEL
LIN {X 0,Y 642.794,Z 832.986,A -85,B 0,C 180,E1 7426.417,E2 7426.417} C_VEL
LIN {X 0,Y 638.667,Z 845.365,A -85,B 0,C 180,E1 7426.338,E2 7426.338} C_VEL
LIN {X 0,Y 632.913,Z 923.896,A -85,B 0,C 180,E1 7428.621,E2 7428.621} C_VEL
LIN {X 0,Y 625.032,Z 997.842,A -85,B 0,C 180,E1 7432.393,E2 7432.393} C_VEL
LIN {X 0,Y 616.898,Z 1062.631,A -85,B 0,C 180,E1 7437.38,E2 7437.38} C_VEL
LIN {X 0,Y 609.904,Z 1118.885,A -85,B 0,C 180,E1 7443.612,E2 7443.612} C_VEL
LIN {X 0,Y 605.797,Z 1162.64,A -85,B 0,C 180,E1 7450.658,E2 7450.658} C_VEL
LIN {X 0,Y 603.707,Z 1192.585,A -85,B 0,C 180,E1 7458.165,E2 7458.165} C_VEL
LIN {X 0,Y 603.045,Z 1206.858,A -85,B 0,C 180,E1 7464.986,E2 7464.986} C_VEL
LIN {X 0,Y 603.039,Z 1209.864,A -85,B 0,C 180,E1 7470.759,E2 7470.759} C_VEL
LIN {X 0,Y 602.955,Z 1203.458,A -85,B 0,C 180,E1 7477.267,E2 7477.267} C_VEL
LIN {X 0,Y 603.487,Z 1187.364,A -85,B 0,C 180,E1 7483.488,E2 7483.488} C_VEL
LIN {X 0,Y 605.333,Z 1160.189,A -85,B 0,C 180,E1 7489.837,E2 7489.837} C_VEL
LIN {X 0,Y 609.691,Z 1118.507,A -85,B 0,C 180,E1 7496.449,E2 7496.449} C_VEL
LIN {X 0,Y 616.69,Z 1062.367,A -85,B 0,C 180,E1 7502.659,E2 7502.659} C_VEL
LIN {X 0,Y 625.436,Z 994.961,A -85,B 0,C 180,E1 7507.786,E2 7507.786} C_VEL
LIN {X 0,Y 633.238,Z 924.569,A -85,B 0,C 180,E1 7511.322,E2 7511.322} C_VEL
LIN {X 0,Y 638.704,Z 849.668,A -85,B 0,C 180,E1 7513.558,E2 7513.558} C_VEL
LIN {X 0,Y 638.162,Z 824.789,A -85,B 0,C 180,E1 7514.137,E2 7514.137} C_VEL
LIN {X 0,Y 602.06,Z 762.06,A -85,B 0,C 180,E1 7518.735,E2 7518.735} C_VEL
LIN {X 0,Y 602.468,Z 762.06,A -85,B 0,C 180,E1 7527.605,E2 7527.605} C_VEL
LIN {X 0,Y 602.555,Z 762.06,A -85,B 0,C 180,E1 7535.404,E2 7535.404} C_VEL
LIN {X 0,Y 602.501,Z 762.06,A -85,B 0,C 180,E1 7544.624,E2 7544.624} C_VEL
LIN {X 0,Y 602.569,Z 762.06,A -85,B 0,C 180,E1 7553.451,E2 7553.451} C_VEL
LIN {X 0,Y 602.804,Z 762.06,A -85,B 0,C 180,E1 7560.679,E2 7560.679} C_VEL
LIN {X 0,Y 602.838,Z 762.06,A -85,B 0,C 180,E1 7567.914,E2 7567.914} C_VEL
LIN {X 0,Y 602.253,Z 762.06,A -85,B 0,C 180,E1 7576.797,E2 7576.797} C_VEL
LIN {X 0,Y 602.336,Z 762.06,A -85,B 0,C 180,E1 7584.512,E2 7584.512} C_VEL
LIN {X 0,Y 602.15,Z 762.06,A -85,B 0,C 180,E1 7592.752,E2 7592.752} C_VEL
LIN {X 0,Y 602.022,Z 762.06,A -85,B 0,C 180,E1 7601.911,E2 7601.911} C_VEL
LIN {X 0,Y 602.4,Z 764.137,A -85,B 0,C 180,E1 7602.927,E2 7602.927} C_VEL
LIN {X 0,Y 638.319,Z 827.841,A -85,B 0,C 180,E1 7606.574,E2 7606.574} C_VEL
LIN {X 0,Y 632.754,Z 898.388,A -85,B 0,C 180,E1 7608.788,E2 7608.788} C_VEL
LIN {X 0,Y 625.003,Z 968.357,A -85,B 0,C 180,E1 7612.387,E2 7612.387} C_VEL
LIN {X 0,Y 616.527,Z 1033.79,A -85,B 0,C 180,E1 7617.427,E2 7617.427} C_VEL
LIN {X 0,Y 609.45,Z 1090.232,A -85,B 0,C 180,E1 7623.726,E2 7623.726} C_VEL
LIN {X 0,Y 605.375,Z 1130.458,A -85,B 0,C 180,E1 7630.182,E2 7630.182} C_VEL
LIN {X 0,Y 603.389,Z 1158.729,A -85,B 0,C 180,E1 7636.88,E2 7636.88} C_VEL
LIN {X 0,Y 602.906,Z 1174.722,A -85,B 0,C 180,E1 7643.459,E2 7643.459} C_VEL
LIN {X 0,Y 602.701,Z 1179.894,A -85,B 0,C 180,E1 7649.24,E2 7649.24} C_VEL
LIN {X 0,Y 602.973,Z 1175.816,A -85,B 0,C 180,E1 7655.739,E2 7655.739} C_VEL
LIN {X 0,Y 603.568,Z 1159.847,A -85,B 0,C 180,E1 7662.668,E2 7662.668} C_VEL
LIN {X 0,Y 605.892,Z 1128.896,A -85,B 0,C 180,E1 7670.012,E2 7670.012} C_VEL
LIN {X 0,Y 610.58,Z 1084.087,A -85,B 0,C 180,E1 7676.957,E2 7676.957} C_VEL
LIN {X 0,Y 617.559,Z 1026.894,A -85,B 0,C 180,E1 7683.095,E2 7683.095} C_VEL
LIN {X 0,Y 625.856,Z 960.692,A -85,B 0,C 180,E1 7688.004,E2 7688.004} C_VEL
LIN {X 0,Y 633.734,Z 887.776,A -85,B 0,C 180,E1 7691.553,E2 7691.553} C_VEL
LIN {X 0,Y 637.15,Z 823.527,A -85,B 0,C 180,E1 7693.543,E2 7693.543} C_VEL
LIN {X 0,Y 602.392,Z 764.105,A -85,B 0,C 180,E1 7696.994,E2 7696.994} C_VEL
LIN {X 0,Y 602.14,Z 762.06,A -85,B 0,C 180,E1 7698.164,E2 7698.164} C_VEL
LIN {X 0,Y 602.923,Z 763.755,A -85,B 0,C 180,E1 7703.838,E2 7703.838} C_VEL
LIN {X 0,Y 608.174,Z 801.471,A -85,B 0,C 180,E1 7705.57,E2 7705.57} C_VEL
LIN {X 0,Y 606.714,Z 856.983,A -85,B 0,C 180,E1 7707.624,E2 7707.624} C_VEL
LIN {X 0,Y 606.798,Z 982.388,A -85,B 0,C 180,E1 7709.394,E2 7709.394} C_VEL
LIN {X 0,Y 606.021,Z 1020.951,A -85,B 0,C 180,E1 7711.325,E2 7711.325} C_VEL
LIN {X 0,Y 604.993,Z 1050.263,A -85,B 0,C 180,E1 7714.291,E2 7714.291} C_VEL
LIN {X 0,Y 604.39,Z 1067.587,A -85,B 0,C 180,E1 7717.916,E2 7717.916} C_VEL
LIN {X 0,Y 604.389,Z 1071.691,A -85,B 0,C 180,E1 7721.756,E2 7721.756} C_VEL
LIN {X 0,Y 604.904,Z 1062.453,A -85,B 0,C 180,E1 7725.584,E2 7725.584} C_VEL
LIN {X 0,Y 605.572,Z 1039.811,A -85,B 0,C 180,E1 7729.029,E2 7729.029} C_VEL
LIN {X 0,Y 606.516,Z 1005.511,A -85,B 0,C 180,E1 7731.6,E2 7731.6} C_VEL
LIN {X 0,Y 606.766,Z 965.34,A -85,B 0,C 180,E1 7732.905,E2 7732.905} C_VEL
LIN {X 0,Y 607.364,Z 845.659,A -85,B 0,C 180,E1 7734.577,E2 7734.577} C_VEL
LIN {X 0,Y 605.991,Z 774.458,A -85,B 0,C 180,E1 7737.51,E2 7737.51} C_VEL
LIN {X 0,Y 603.078,Z 762.06,A -85,B 0,C 180,E1 7738.24,E2 7738.24} C_VEL
LIN {X 0,Y 602.667,Z 762.06,A -85,B 0,C 180,E1 7746.548,E2 7746.548} C_VEL
LIN {X 0,Y 602.26,Z 762.06,A -85,B 0,C 180,E1 7755.382,E2 7755.382} C_VEL
LIN {X 0,Y 602.07,Z 762.06,A -85,B 0,C 180,E1 7763.19,E2 7763.19} C_VEL
LIN {X 0,Y 602.089,Z 762.06,A -85,B 0,C 180,E1 7771.154,E2 7771.154} C_VEL
LIN {X 0,Y 601.823,Z 762.06,A -85,B 0,C 180,E1 7780.062,E2 7780.062} C_VEL
LIN {X 0,Y 602.062,Z 763.991,A -85,B 0,C 180,E1 7781.369,E2 7781.369} C_VEL
LIN {X 0,Y 639.279,Z 827.1,A -85,B 0,C 180,E1 7786.004,E2 7786.004} C_VEL
LIN {X 0,Y 638.667,Z 845.365,A -85,B 0,C 180,E1 7786.338,E2 7786.338} C_VEL
LIN {X 0,Y 631.053,Z 879.854,A -85,B 0,C 180,E1 7786.68,E2 7786.68} C_VEL
LIN {X 0,Y 624.187,Z 951.626,A -85,B 0,C 180,E1 7789.367,E2 7789.367} C_VEL
LIN {X 0,Y 615.1,Z 1023.24,A -85,B 0,C 180,E1 7793.667,E2 7793.667} C_VEL
LIN {X 0,Y 606.656,Z 1085.178,A -85,B 0,C 180,E1 7799.198,E2 7799.198} C_VEL
LIN {X 0,Y 600.117,Z 1136.59,A -85,B 0,C 180,E1 7805.809,E2 7805.809} C_VEL
LIN {X 0,Y 596.675,Z 1173.037,A -85,B 0,C 180,E1 7812.614,E2 7812.614} C_VEL
LIN {X 0,Y 595.351,Z 1195.597,A -85,B 0,C 180,E1 7819.088,E2 7819.088} C_VEL
LIN {X 0,Y 595.075,Z 1206.857,A -85,B 0,C 180,E1 7824.919,E2 7824.919} C_VEL
LIN {X 0,Y 595.062,Z 1209.864,A -85,B 0,C 180,E1 7830.769,E2 7830.769} C_VEL
LIN {X 0,Y 594.977,Z 1203.458,A -85,B 0,C 180,E1 7837.365,E2 7837.365} C_VEL
LIN {X 0,Y 595.598,Z 1186.047,A -85,B 0,C 180,E1 7844.046,E2 7844.046} C_VEL
LIN {X 0,Y 597.719,Z 1158.312,A -85,B 0,C 180,E1 7850.47,E2 7850.47} C_VEL
LIN {X 0,Y 602.359,Z 1116.827,A -85,B 0,C 180,E1 7857.026,E2 7857.026} C_VEL
LIN {X 0,Y 609.958,Z 1060.211,A -85,B 0,C 180,E1 7863.285,E2 7863.285} C_VEL
LIN {X 0,Y 619.199,Z 992.664,A -85,B 0,C 180,E1 7868.396,E2 7868.396} C_VEL
LIN {X 0,Y 627.205,Z 923.962,A -85,B 0,C 180,E1 7871.836,E2 7871.836} C_VEL
LIN {X 0,Y 632.84,Z 850.508,A -85,B 0,C 180,E1 7874.042,E2 7874.042} C_VEL
LIN {X 0,Y 632.347,Z 828.282,A -85,B 0,C 180,E1 7874.58,E2 7874.58} C_VEL
LIN {X 0,Y 594.085,Z 762.06,A -85,B 0,C 180,E1 7879.686,E2 7879.686} C_VEL
LIN {X 0,Y 594.514,Z 762.06,A -85,B 0,C 180,E1 7888.834,E2 7888.834} C_VEL
LIN {X 0,Y 594.379,Z 762.06,A -85,B 0,C 180,E1 7896.646,E2 7896.646} C_VEL
LIN {X 0,Y 594.396,Z 762.06,A -85,B 0,C 180,E1 7905.922,E2 7905.922} C_VEL
LIN {X 0,Y 594.58,Z 762.06,A -85,B 0,C 180,E1 7913.363,E2 7913.363} C_VEL
LIN {X 0,Y 594.804,Z 762.06,A -85,B 0,C 180,E1 7920.688,E2 7920.688} C_VEL
LIN {X 0,Y 594.788,Z 762.06,A -85,B 0,C 180,E1 7928.022,E2 7928.022} C_VEL
LIN {X 0,Y 594.205,Z 762.06,A -85,B 0,C 180,E1 7937.031,E2 7937.031} C_VEL
LIN {X 0,Y 594.282,Z 762.06,A -85,B 0,C 180,E1 7944.896,E2 7944.896} C_VEL
LIN {X 0,Y 594.036,Z 762.06,A -85,B 0,C 180,E1 7953.817,E2 7953.817} C_VEL
LIN {X 0,Y 594.24,Z 763.729,A -85,B 0,C 180,E1 7962.324,E2 7962.324} C_VEL
LIN {X 0,Y 632.069,Z 834.428,A -85,B 0,C 180,E1 7966.238,E2 7966.238} C_VEL
LIN {X 0,Y 626.124,Z 903.68,A -85,B 0,C 180,E1 7968.516,E2 7968.516} C_VEL
LIN {X 0,Y 617.863,Z 972.572,A -85,B 0,C 180,E1 7972.195,E2 7972.195} C_VEL
LIN {X 0,Y 608.907,Z 1037.739,A -85,B 0,C 180,E1 7977.386,E2 7977.386} C_VEL
LIN {X 0,Y 601.59,Z 1092.987,A -85,B 0,C 180,E1 7983.765,E2 7983.765} C_VEL
LIN {X 0,Y 597.378,Z 1132.437,A -85,B 0,C 180,E1 7990.292,E2 7990.292} C_VEL
LIN {X 0,Y 595.37,Z 1159.877,A -85,B 0,C 180,E1 7997.075,E2 7997.075} C_VEL
LIN {X 0,Y 594.945,Z 1174.718,A -85,B 0,C 180,E1 8003.371,E2 8003.371} C_VEL
LIN {X 0,Y 594.703,Z 1179.896,A -85,B 0,C 180,E1 8009.23,E2 8009.23} C_VEL
LIN {X 0,Y 594.996,Z 1175.814,A -85,B 0,C 180,E1 8015.816,E2 8015.816} C_VEL
LIN {X 0,Y 595.666,Z 1159.845,A -85,B 0,C 180,E1 8022.839,E2 8022.839} C_VEL
LIN {X 0,Y 598.171,Z 1128.899,A -85,B 0,C 180,E1 8030.282,E2 8030.282} C_VEL
LIN {X 0,Y 603.219,Z 1083.487,A -85,B 0,C 180,E1 8037.395,E2 8037.395} C_VEL
LIN {X 0,Y 610.58,Z 1026.904,A -85,B 0,C 180,E1 8043.522,E2 8043.522} C_VEL
LIN {X 0,Y 619.352,Z 960.696,A -85,B 0,C 180,E1 8048.475,E2 8048.475} C_VEL
LIN {X 0,Y 627.686,Z 887.281,A -85,B 0,C 180,E1 8052.066,E2 8052.066} C_VEL
LIN {X 0,Y 631.185,Z 826.895,A -85,B 0,C 180,E1 8053.958,E2 8053.958} C_VEL
LIN {X 0,Y 594.527,Z 764.594,A -85,B 0,C 180,E1 8057.548,E2 8057.548} C_VEL
LIN {X 0,Y 594.117,Z 762.06,A -85,B 0,C 180,E1 8057.822,E2 8057.822} C_VEL
LIN {X 0,Y 594.764,Z 763.337,A -85,B 0,C 180,E1 8063.581,E2 8063.581} C_VEL
LIN {X 0,Y 600.42,Z 802.584,A -85,B 0,C 180,E1 8065.401,E2 8065.401} C_VEL
LIN {X 0,Y 598.927,Z 856.399,A -85,B 0,C 180,E1 8067.443,E2 8067.443} C_VEL
LIN {X 0,Y 598.989,Z 983.117,A -85,B 0,C 180,E1 8069.252,E2 8069.252} C_VEL
LIN {X 0,Y 598.161,Z 1022.391,A -85,B 0,C 180,E1 8071.242,E2 8071.242} C_VEL
LIN {X 0,Y 597.124,Z 1052.201,A -85,B 0,C 180,E1 8074.343,E2 8074.343} C_VEL
LIN {X 0,Y 596.492,Z 1069.196,A -85,B 0,C 180,E1 8078.094,E2 8078.094} C_VEL
LIN {X 0,Y 596.455,Z 1072.898,A -85,B 0,C 180,E1 8081.505,E2 8081.505} C_VEL
LIN {X 0,Y 596.918,Z 1064.424,A -85,B 0,C 180,E1 8085.443,E2 8085.443} C_VEL
LIN {X 0,Y 597.737,Z 1043.041,A -85,B 0,C 180,E1 8088.895,E2 8088.895} C_VEL
LIN {X 0,Y 598.71,Z 1009.304,A -85,B 0,C 180,E1 8091.573,E2 8091.573} C_VEL
LIN {X 0,Y 598.933,Z 968.739,A -85,B 0,C 180,E1 8092.995,E2 8092.995} C_VEL
LIN {X 0,Y 599.62,Z 846.787,A -85,B 0,C 180,E1 8094.734,E2 8094.734} C_VEL
LIN {X 0,Y 598.178,Z 775.546,A -85,B 0,C 180,E1 8097.691,E2 8097.691} C_VEL
LIN {X 0,Y 595.006,Z 762.06,A -85,B 0,C 180,E1 8098.399,E2 8098.399} C_VEL
LIN {X 0,Y 594.631,Z 762.06,A -85,B 0,C 180,E1 8106.636,E2 8106.636} C_VEL
LIN {X 0,Y 594.508,Z 762.06,A -85,B 0,C 180,E1 8114.075,E2 8114.075} C_VEL
LIN {X 0,Y 594.046,Z 762.06,A -85,B 0,C 180,E1 8123.368,E2 8123.368} C_VEL
LIN {X 0,Y 594.02,Z 762.06,A -85,B 0,C 180,E1 8131.625,E2 8131.625} C_VEL
LIN {X 0,Y 593.864,Z 762.664,A -85,B 0,C 180,E1 8140.443,E2 8140.443} C_VEL
LIN {X 0,Y 633.608,Z 830.764,A -85,B 0,C 180,E1 8145.58,E2 8145.58} C_VEL
LIN {X 0,Y 631.053,Z 879.854,A -85,B 0,C 180,E1 8146.68,E2 8146.68} C_VEL
LIN {X 0,Y 621.978,Z 913.632,A -85,B 0,C 180,E1 8147.246,E2 8147.246} C_VEL
LIN {X 0,Y 613.467,Z 987.438,A -85,B 0,C 180,E1 8150.809,E2 8150.809} C_VEL
LIN {X 0,Y 603.962,Z 1054.083,A -85,B 0,C 180,E1 8155.733,E2 8155.733} C_VEL
LIN {X 0,Y 595.64,Z 1111.683,A -85,B 0,C 180,E1 8161.927,E2 8161.927} C_VEL
LIN {X 0,Y 590.35,Z 1156.753,A -85,B 0,C 180,E1 8168.952,E2 8168.952} C_VEL
LIN {X 0,Y 588.115,Z 1188.836,A -85,B 0,C 180,E1 8176.614,E2 8176.614} C_VEL
LIN {X 0,Y 587.51,Z 1204.811,A -85,B 0,C 180,E1 8183.366,E2 8183.366} C_VEL
LIN {X 0,Y 587.057,Z 1209.864,A -85,B 0,C 180,E1 8190.78,E2 8190.78} C_VEL
LIN {X 0,Y 586.978,Z 1203.459,A -85,B 0,C 180,E1 8197.466,E2 8197.466} C_VEL
LIN {X 0,Y 587.702,Z 1186.047,A -85,B 0,C 180,E1 8204.238,E2 8204.238} C_VEL
LIN {X 0,Y 590.119,Z 1156.333,A -85,B 0,C 180,E1 8211.14,E2 8211.14} C_VEL
LIN {X 0,Y 595.777,Z 1111.055,A -85,B 0,C 180,E1 8218.154,E2 8218.154} C_VEL
LIN {X 0,Y 604.065,Z 1053.358,A -85,B 0,C 180,E1 8224.332,E2 8224.332} C_VEL
LIN {X 0,Y 613.547,Z 986.295,A -85,B 0,C 180,E1 8229.266,E2 8229.266} C_VEL
LIN {X 0,Y 621.873,Z 916.732,A -85,B 0,C 180,E1 8232.617,E2 8232.617} C_VEL
LIN {X 0,Y 627.462,Z 843.165,A -85,B 0,C 180,E1 8234.682,E2 8234.682} C_VEL
LIN {X 0,Y 625.994,Z 830.491,A -85,B 0,C 180,E1 8235.1,E2 8235.1} C_VEL
LIN {X 0,Y 588.397,Z 767.664,A -85,B 0,C 180,E1 8240.094,E2 8240.094} C_VEL
LIN {X 0,Y 586.147,Z 762.06,A -85,B 0,C 180,E1 8240.584,E2 8240.584} C_VEL
LIN {X 0,Y 586.488,Z 762.06,A -85,B 0,C 180,E1 8250.156,E2 8250.156} C_VEL
LIN {X 0,Y 586.182,Z 762.06,A -85,B 0,C 180,E1 8257.909,E2 8257.909} C_VEL
LIN {X 0,Y 586.371,Z 762.06,A -85,B 0,C 180,E1 8266.183,E2 8266.183} C_VEL
LIN {X 0,Y 586.425,Z 762.06,A -85,B 0,C 180,E1 8274.761,E2 8274.761} C_VEL
LIN {X 0,Y 586.796,Z 762.06,A -85,B 0,C 180,E1 8280.697,E2 8280.697} C_VEL
LIN {X 0,Y 586.74,Z 762.06,A -85,B 0,C 180,E1 8288.133,E2 8288.133} C_VEL
LIN {X 0,Y 586.153,Z 762.06,A -85,B 0,C 180,E1 8297.273,E2 8297.273} C_VEL
LIN {X 0,Y 586.261,Z 762.06,A -85,B 0,C 180,E1 8305.231,E2 8305.231} C_VEL
LIN {X 0,Y 586.06,Z 762.06,A -85,B 0,C 180,E1 8313.77,E2 8313.77} C_VEL
LIN {X 0,Y 586.12,Z 763.401,A -85,B 0,C 180,E1 8321.595,E2 8321.595} C_VEL
LIN {X 0,Y 625.53,Z 836.414,A -85,B 0,C 180,E1 8325.844,E2 8325.844} C_VEL
LIN {X 0,Y 620.361,Z 900.367,A -85,B 0,C 180,E1 8327.879,E2 8327.879} C_VEL
LIN {X 0,Y 611.739,Z 969.934,A -85,B 0,C 180,E1 8331.547,E2 8331.547} C_VEL
LIN {X 0,Y 602.294,Z 1035.087,A -85,B 0,C 180,E1 8336.698,E2 8336.698} C_VEL
LIN {X 0,Y 594.509,Z 1090.298,A -85,B 0,C 180,E1 8343.025,E2 8343.025} C_VEL
LIN {X 0,Y 589.56,Z 1132.902,A -85,B 0,C 180,E1 8350.113,E2 8350.113} C_VEL
LIN {X 0,Y 587.443,Z 1159.872,A -85,B 0,C 180,E1 8356.898,E2 8356.898} C_VEL
LIN {X 0,Y 586.956,Z 1174.715,A -85,B 0,C 180,E1 8363.28,E2 8363.28} C_VEL
LIN {X 0,Y 586.704,Z 1179.899,A -85,B 0,C 180,E1 8369.22,E2 8369.22} C_VEL
LIN {X 0,Y 586.937,Z 1176.836,A -85,B 0,C 180,E1 8375.152,E2 8375.152} C_VEL
LIN {X 0,Y 587.311,Z 1163.243,A -85,B 0,C 180,E1 8381.888,E2 8381.888} C_VEL
LIN {X 0,Y 589.132,Z 1137.839,A -85,B 0,C 180,E1 8388.739,E2 8388.739} C_VEL
LIN {X 0,Y 593.507,Z 1098.405,A -85,B 0,C 180,E1 8395.718,E2 8395.718} C_VEL
LIN {X 0,Y 600.772,Z 1045.618,A -85,B 0,C 180,E1 8402.173,E2 8402.173} C_VEL
LIN {X 0,Y 610.083,Z 981.682,A -85,B 0,C 180,E1 8407.586,E2 8407.586} C_VEL
LIN {X 0,Y 619.095,Z 912.269,A -85,B 0,C 180,E1 8411.514,E2 8411.514} C_VEL
LIN {X 0,Y 625.144,Z 845.898,A -85,B 0,C 180,E1 8413.838,E2 8413.838} C_VEL
LIN {X 0,Y 624.043,Z 829.224,A -85,B 0,C 180,E1 8414.356,E2 8414.356} C_VEL
LIN {X 0,Y 588.842,Z 768.422,A -85,B 0,C 180,E1 8417.948,E2 8417.948} C_VEL
LIN {X 0,Y 586.163,Z 762.06,A -85,B 0,C 180,E1 8418.447,E2 8418.447} C_VEL
LIN {X 0,Y 586.838,Z 763.853,A -85,B 0,C 180,E1 8423.359,E2 8423.359} C_VEL
LIN {X 0,Y 592.707,Z 804.619,A -85,B 0,C 180,E1 8425.268,E2 8425.268} C_VEL
LIN {X 0,Y 591.145,Z 859.65,A -85,B 0,C 180,E1 8427.307,E2 8427.307} C_VEL
LIN {X 0,Y 591.177,Z 984.768,A -85,B 0,C 180,E1 8429.133,E2 8429.133} C_VEL
LIN {X 0,Y 590.322,Z 1023.737,A -85,B 0,C 180,E1 8431.152,E2 8431.152} C_VEL
LIN {X 0,Y 589.237,Z 1053.345,A -85,B 0,C 180,E1 8434.279,E2 8434.279} C_VEL
LIN {X 0,Y 588.594,Z 1070.364,A -85,B 0,C 180,E1 8438.098,E2 8438.098} C_VEL
LIN {X 0,Y 588.544,Z 1074.088,A -85,B 0,C 180,E1 8441.247,E2 8441.247} C_VEL
LIN {X 0,Y 589.007,Z 1065.911,A -85,B 0,C 180,E1 8445.409,E2 8445.409} C_VEL
LIN {X 0,Y 589.873,Z 1044.709,A -85,B 0,C 180,E1 8448.921,E2 8448.921} C_VEL
LIN {X 0,Y 590.846,Z 1011.945,A -85,B 0,C 180,E1 8451.603,E2 8451.603} C_VEL
LIN {X 0,Y 591.112,Z 972.099,A -85,B 0,C 180,E1 8453.087,E2 8453.087} C_VEL
LIN {X 0,Y 591.874,Z 848.058,A -85,B 0,C 180,E1 8454.896,E2 8454.896} C_VEL
LIN {X 0,Y 590.505,Z 777.407,A -85,B 0,C 180,E1 8457.834,E2 8457.834} C_VEL
LIN {X 0,Y 586.835,Z 762.06,A -85,B 0,C 180,E1 8458.747,E2 8458.747} C_VEL
LIN {X 0,Y 586.606,Z 762.06,A -85,B 0,C 180,E1 8466.728,E2 8466.728} C_VEL
LIN {X 0,Y 586.469,Z 762.06,A -85,B 0,C 180,E1 8474.272,E2 8474.272} C_VEL
LIN {X 0,Y 586.056,Z 762.06,A -85,B 0,C 180,E1 8483.302,E2 8483.302} C_VEL
LIN {X 0,Y 585.936,Z 762.06,A -85,B 0,C 180,E1 8492.113,E2 8492.113} C_VEL
LIN {X 0,Y 585.976,Z 763.555,A -85,B 0,C 180,E1 8499.55,E2 8499.55} C_VEL
LIN {X 0,Y 624.883,Z 828.451,A -85,B 0,C 180,E1 8504.756,E2 8504.756} C_VEL
LIN {X 0,Y 627.344,Z 839.576,A -85,B 0,C 180,E1 8505.222,E2 8505.222} C_VEL
LIN {X 0,Y 621.978,Z 913.632,A -85,B 0,C 180,E1 8507.246,E2 8507.246} C_VEL
LIN {X 0,Y 612.394,Z 946.429,A -85,B 0,C 180,E1 8508.118,E2 8508.118} C_VEL
LIN {X 0,Y 602.875,Z 1016.068,A -85,B 0,C 180,E1 8512.208,E2 8512.208} C_VEL
LIN {X 0,Y 593.54,Z 1077.609,A -85,B 0,C 180,E1 8517.572,E2 8517.572} C_VEL
LIN {X 0,Y 586.111,Z 1130.28,A -85,B 0,C 180,E1 8524.171,E2 8524.171} C_VEL
LIN {X 0,Y 581.326,Z 1171.587,A -85,B 0,C 180,E1 8531.789,E2 8531.789} C_VEL
LIN {X 0,Y 579.485,Z 1195.409,A -85,B 0,C 180,E1 8538.715,E2 8538.715} C_VEL
LIN {X 0,Y 579.138,Z 1206.854,A -85,B 0,C 180,E1 8544.779,E2 8544.779} C_VEL
LIN {X 0,Y 579.052,Z 1209.864,A -85,B 0,C 180,E1 8550.791,E2 8550.791} C_VEL
LIN {X 0,Y 578.995,Z 1203.459,A -85,B 0,C 180,E1 8557.569,E2 8557.569} C_VEL
LIN {X 0,Y 579.792,Z 1186.046,A -85,B 0,C 180,E1 8564.437,E2 8564.437} C_VEL
LIN {X 0,Y 582.371,Z 1156.335,A -85,B 0,C 180,E1 8571.435,E2 8571.435} C_VEL
LIN {X 0,Y 588.397,Z 1111.056,A -85,B 0,C 180,E1 8578.539,E2 8578.539} C_VEL
LIN {X 0,Y 597.158,Z 1053.558,A -85,B 0,C 180,E1 8584.765,E2 8584.765} C_VEL
LIN {X 0,Y 607.107,Z 986.799,A -85,B 0,C 180,E1 8589.728,E2 8589.728} C_VEL
LIN {X 0,Y 615.632,Z 918.103,A -85,B 0,C 180,E1 8593.063,E2 8593.063} C_VEL
LIN {X 0,Y 621.541,Z 845.187,A -85,B 0,C 180,E1 8595.155,E2 8595.155} C_VEL
LIN {X 0,Y 619.94,Z 833.339,A -85,B 0,C 180,E1 8595.592,E2 8595.592} C_VEL
LIN {X 0,Y 583.693,Z 772.667,A -85,B 0,C 180,E1 8600.557,E2 8600.557} C_VEL
LIN {X 0,Y 578.103,Z 762.06,A -85,B 0,C 180,E1 8601.582,E2 8601.582} C_VEL
LIN {X 0,Y 578.441,Z 762.06,A -85,B 0,C 180,E1 8610.92,E2 8610.92} C_VEL
LIN {X 0,Y 578.073,Z 762.06,A -85,B 0,C 180,E1 8619.2,E2 8619.2} C_VEL
LIN {X 0,Y 578.261,Z 762.06,A -85,B 0,C 180,E1 8627.068,E2 8627.068} C_VEL
LIN {X 0,Y 578.426,Z 762.06,A -85,B 0,C 180,E1 8634.688,E2 8634.688} C_VEL
LIN {X 0,Y 578.789,Z 762.06,A -85,B 0,C 180,E1 8640.707,E2 8640.707} C_VEL
LIN {X 0,Y 578.694,Z 762.06,A -85,B 0,C 180,E1 8648.247,E2 8648.247} C_VEL
LIN {X 0,Y 578.107,Z 762.06,A -85,B 0,C 180,E1 8657.521,E2 8657.521} C_VEL
LIN {X 0,Y 578.232,Z 762.06,A -85,B 0,C 180,E1 8665.606,E2 8665.606} C_VEL
LIN {X 0,Y 578.037,Z 762.06,A -85,B 0,C 180,E1 8674.303,E2 8674.303} C_VEL
LIN {X 0,Y 578.182,Z 763.982,A -85,B 0,C 180,E1 8680.82,E2 8680.82} C_VEL
LIN {X 0,Y 618.729,Z 839.525,A -85,B 0,C 180,E1 8685.496,E2 8685.496} C_VEL
LIN {X 0,Y 612.975,Z 912.085,A -85,B 0,C 180,E1 8687.886,E2 8687.886} C_VEL
LIN {X 0,Y 603.916,Z 979.241,A -85,B 0,C 180,E1 8691.682,E2 8691.682} C_VEL
LIN {X 0,Y 593.993,Z 1043.161,A -85,B 0,C 180,E1 8697.057,E2 8697.057} C_VEL
LIN {X 0,Y 586.178,Z 1095.889,A -85,B 0,C 180,E1 8703.464,E2 8703.464} C_VEL
LIN {X 0,Y 581.525,Z 1134.897,A -85,B 0,C 180,E1 8710.255,E2 8710.255} C_VEL
LIN {X 0,Y 579.392,Z 1161.006,A -85,B 0,C 180,E1 8717.097,E2 8717.097} C_VEL
LIN {X 0,Y 578.965,Z 1175.708,A -85,B 0,C 180,E1 8723.863,E2 8723.863} C_VEL
LIN {X 0,Y 579.048,Z 1179.899,A -85,B 0,C 180,E1 8730.711,E2 8730.711} C_VEL
LIN {X 0,Y 579.502,Z 1172.094,A -85,B 0,C 180,E1 8738.24,E2 8738.24} C_VEL
LIN {X 0,Y 580.395,Z 1150.762,A -85,B 0,C 180,E1 8745.891,E2 8745.891} C_VEL
LIN {X 0,Y 583.706,Z 1116.536,A -85,B 0,C 180,E1 8753.156,E2 8753.156} C_VEL
LIN {X 0,Y 590.191,Z 1068.595,A -85,B 0,C 180,E1 8760.043,E2 8760.043} C_VEL
LIN {X 0,Y 599.561,Z 1007.833,A -85,B 0,C 180,E1 8766.068,E2 8766.068} C_VEL
LIN {X 0,Y 609.577,Z 938.801,A -85,B 0,C 180,E1 8770.704,E2 8770.704} C_VEL
LIN {X 0,Y 616.022,Z 874.336,A -85,B 0,C 180,E1 8773.46,E2 8773.46} C_VEL
LIN {X 0,Y 617.828,Z 833.354,A -85,B 0,C 180,E1 8774.645,E2 8774.645} C_VEL
LIN {X 0,Y 578.227,Z 763.14,A -85,B 0,C 180,E1 8779.108,E2 8779.108} C_VEL
LIN {X 0,Y 578.602,Z 762.827,A -85,B 0,C 180,E1 8783.048,E2 8783.048} C_VEL
LIN {X 0,Y 585.011,Z 805.448,A -85,B 0,C 180,E1 8785.079,E2 8785.079} C_VEL
LIN {X 0,Y 583.394,Z 858.562,A -85,B 0,C 180,E1 8787.109,E2 8787.109} C_VEL
LIN {X 0,Y 583.364,Z 984.698,A -85,B 0,C 180,E1 8788.96,E2 8788.96} C_VEL
LIN {X 0,Y 582.508,Z 1023.643,A -85,B 0,C 180,E1 8790.954,E2 8790.954} C_VEL
LIN {X 0,Y 581.357,Z 1053.891,A -85,B 0,C 180,E1 8794.126,E2 8794.126} C_VEL
LIN {X 0,Y 580.687,Z 1071.187,A -85,B 0,C 180,E1 8797.96,E2 8797.96} C_VEL
LIN {X 0,Y 580.675,Z 1074.5,A -85,B 0,C 180,E1 8802.377,E2 8802.377} C_VEL
LIN {X 0,Y 581.455,Z 1062.616,A -85,B 0,C 180,E1 8806.463,E2 8806.463} C_VEL
LIN {X 0,Y 582.123,Z 1037.439,A -85,B 0,C 180,E1 8809.912,E2 8809.912} C_VEL
LIN {X 0,Y 583.118,Z 1000.35,A -85,B 0,C 180,E1 8812.381,E2 8812.381} C_VEL
LIN {X 0,Y 583.204,Z 954.316,A -85,B 0,C 180,E1 8813.508,E2 8813.508} C_VEL
LIN {X 0,Y 584.141,Z 849.1,A -85,B 0,C 180,E1 8815.061,E2 8815.061} C_VEL
LIN {X 0,Y 582.844,Z 779.157,A -85,B 0,C 180,E1 8817.992,E2 8817.992} C_VEL
LIN {X 0,Y 578.764,Z 762.06,A -85,B 0,C 180,E1 8818.917,E2 8818.917} C_VEL
LIN {X 0,Y 578.572,Z 762.06,A -85,B 0,C 180,E1 8826.822,E2 8826.822} C_VEL
LIN {X 0,Y 578.406,Z 762.06,A -85,B 0,C 180,E1 8834.476,E2 8834.476} C_VEL
LIN {X 0,Y 578.12,Z 762.06,A -85,B 0,C 180,E1 8842.415,E2 8842.415} C_VEL
LIN {X 0,Y 577.943,Z 762.06,A -85,B 0,C 180,E1 8851.509,E2 8851.509} C_VEL
LIN {X 0,Y 577.975,Z 763.711,A -85,B 0,C 180,E1 8858.586,E2 8858.586} C_VEL
LIN {X 0,Y 617.494,Z 828.63,A -85,B 0,C 180,E1 8864.077,E2 8864.077} C_VEL
LIN {X 0,Y 621.476,Z 841.542,A -85,B 0,C 180,E1 8864.746,E2 8864.746} C_VEL
LIN {X 0,Y 614.742,Z 923.195,A -85,B 0,C 180,E1 8867.103,E2 8867.103} C_VEL
LIN {X 0,Y 612.394,Z 946.429,A -85,B 0,C 180,E1 8868.118,E2 8868.118} C_VEL
LIN {X 0,Y 602.144,Z 978.151,A -85,B 0,C 180,E1 8869.266,E2 8869.266} C_VEL
LIN {X 0,Y 591.723,Z 1044.844,A -85,B 0,C 180,E1 8873.991,E2 8873.991} C_VEL
LIN {X 0,Y 582.015,Z 1103.858,A -85,B 0,C 180,E1 8880.139,E2 8880.139} C_VEL
LIN {X 0,Y 575.444,Z 1149.802,A -85,B 0,C 180,E1 8887.035,E2 8887.035} C_VEL
LIN {X 0,Y 572.246,Z 1180.901,A -85,B 0,C 180,E1 8893.877,E2 8893.877} C_VEL
LIN {X 0,Y 571.109,Z 1200.727,A -85,B 0,C 180,E1 8900.868,E2 8900.868} C_VEL
LIN {X 0,Y 571.136,Z 1209.399,A -85,B 0,C 180,E1 8907.757,E2 8907.757} C_VEL
LIN {X 0,Y 571.35,Z 1206.754,A -85,B 0,C 180,E1 8915.374,E2 8915.374} C_VEL
LIN {X 0,Y 571.596,Z 1192.068,A -85,B 0,C 180,E1 8922.692,E2 8922.692} C_VEL
LIN {X 0,Y 573.59,Z 1166.224,A -85,B 0,C 180,E1 8929.687,E2 8929.687} C_VEL
LIN {X 0,Y 578.665,Z 1126.387,A -85,B 0,C 180,E1 8936.789,E2 8936.789} C_VEL
LIN {X 0,Y 587.227,Z 1072.271,A -85,B 0,C 180,E1 8943.438,E2 8943.438} C_VEL
LIN {X 0,Y 597.914,Z 1006.339,A -85,B 0,C 180,E1 8948.966,E2 8948.966} C_VEL
LIN {X 0,Y 607.27,Z 938.386,A -85,B 0,C 180,E1 8952.736,E2 8952.736} C_VEL
LIN {X 0,Y 614.64,Z 859.776,A -85,B 0,C 180,E1 8955.37,E2 8955.37} C_VEL
LIN {X 0,Y 614.623,Z 837.741,A -85,B 0,C 180,E1 8955.972,E2 8955.972} C_VEL
LIN {X 0,Y 577.598,Z 774.836,A -85,B 0,C 180,E1 8961.256,E2 8961.256} C_VEL
LIN {X 0,Y 570.125,Z 762.06,A -85,B 0,C 180,E1 8962.63,E2 8962.63} C_VEL
LIN {X 0,Y 570.449,Z 762.06,A -85,B 0,C 180,E1 8972.21,E2 8972.21} C_VEL
LIN {X 0,Y 570.275,Z 762.06,A -85,B 0,C 180,E1 8982.137,E2 8982.137} C_VEL
LIN {X 0,Y 570.856,Z 762.06,A -85,B 0,C 180,E1 8991.549,E2 8991.549} C_VEL
LIN {X 0,Y 570.782,Z 762.06,A -85,B 0,C 180,E1 9000.717,E2 9000.717} C_VEL
LIN {X 0,Y 570.677,Z 762.06,A -85,B 0,C 180,E1 9008.363,E2 9008.363} C_VEL
LIN {X 0,Y 570.333,Z 762.06,A -85,B 0,C 180,E1 9016.174,E2 9016.174} C_VEL
LIN {X 0,Y 570.27,Z 762.06,A -85,B 0,C 180,E1 9024.306,E2 9024.306} C_VEL
LIN {X 0,Y 570.019,Z 762.06,A -85,B 0,C 180,E1 9033.016,E2 9033.016} C_VEL
LIN {X 0,Y 570.225,Z 764.054,A -85,B 0,C 180,E1 9039.97,E2 9039.97} C_VEL
LIN {X 0,Y 610.501,Z 837.47,A -85,B 0,C 180,E1 9044.918,E2 9044.918} C_VEL
LIN {X 0,Y 605.872,Z 915.564,A -85,B 0,C 180,E1 9047.619,E2 9047.619} C_VEL
LIN {X 0,Y 598.152,Z 974.379,A -85,B 0,C 180,E1 9050.862,E2 9050.862} C_VEL
LIN {X 0,Y 587.614,Z 1039.341,A -85,B 0,C 180,E1 9056.23,E2 9056.23} C_VEL
LIN {X 0,Y 578.994,Z 1094.097,A -85,B 0,C 180,E1 9062.833,E2 9062.833} C_VEL
LIN {X 0,Y 573.81,Z 1134.589,A -85,B 0,C 180,E1 9069.908,E2 9069.908} C_VEL
LIN {X 0,Y 571.46,Z 1161,A -85,B 0,C 180,E1 9076.915,E2 9076.915} C_VEL
LIN {X 0,Y 570.996,Z 1175.933,A -85,B 0,C 180,E1 9083.934,E2 9083.934} C_VEL
LIN {X 0,Y 571.047,Z 1179.902,A -85,B 0,C 180,E1 9090.721,E2 9090.721} C_VEL
LIN {X 0,Y 571.507,Z 1172.092,A -85,B 0,C 180,E1 9098.356,E2 9098.356} C_VEL
LIN {X 0,Y 572.429,Z 1150.766,A -85,B 0,C 180,E1 9106.118,E2 9106.118} C_VEL
LIN {X 0,Y 576.012,Z 1116.202,A -85,B 0,C 180,E1 9113.547,E2 9113.547} C_VEL
LIN {X 0,Y 582.901,Z 1068.597,A -85,B 0,C 180,E1 9120.458,E2 9120.458} C_VEL
LIN {X 0,Y 592.734,Z 1008.461,A -85,B 0,C 180,E1 9126.491,E2 9126.491} C_VEL
LIN {X 0,Y 602.941,Z 941.367,A -85,B 0,C 180,E1 9131.064,E2 9131.064} C_VEL
LIN {X 0,Y 610.159,Z 865.433,A -85,B 0,C 180,E1 9134.159,E2 9134.159} C_VEL
LIN {X 0,Y 610.845,Z 836.078,A -85,B 0,C 180,E1 9135.014,E2 9135.014} C_VEL
LIN {X 0,Y 578.957,Z 779.222,A -85,B 0,C 180,E1 9138.625,E2 9138.625} C_VEL
LIN {X 0,Y 570.232,Z 762.06,A -85,B 0,C 180,E1 9140.042,E2 9140.042} C_VEL
LIN {X 0,Y 570.561,Z 763.047,A -85,B 0,C 180,E1 9142.796,E2 9142.796} C_VEL
LIN {X 0,Y 577.319,Z 805.02,A -85,B 0,C 180,E1 9144.829,E2 9144.829} C_VEL
LIN {X 0,Y 575.633,Z 861.488,A -85,B 0,C 180,E1 9146.959,E2 9146.959} C_VEL
LIN {X 0,Y 575.553,Z 986.828,A -85,B 0,C 180,E1 9148.849,E2 9148.849} C_VEL
LIN {X 0,Y 574.666,Z 1025.724,A -85,B 0,C 180,E1 9150.912,E2 9150.912} C_VEL
LIN {X 0,Y 573.473,Z 1055.75,A -85,B 0,C 180,E1 9154.166,E2 9154.166} C_VEL
LIN {X 0,Y 572.77,Z 1071.828,A -85,B 0,C 180,E1 9157.74,E2 9157.74} C_VEL
LIN {X 0,Y 572.737,Z 1076.219,A -85,B 0,C 180,E1 9161.511,E2 9161.511} C_VEL
LIN {X 0,Y 573.215,Z 1068.292,A -85,B 0,C 180,E1 9165.482,E2 9165.482} C_VEL
LIN {X 0,Y 574.178,Z 1046.273,A -85,B 0,C 180,E1 9169.193,E2 9169.193} C_VEL
LIN {X 0,Y 575.243,Z 1011.912,A -85,B 0,C 180,E1 9171.99,E2 9171.99} C_VEL
LIN {X 0,Y 575.481,Z 971.613,A -85,B 0,C 180,E1 9173.421,E2 9173.421} C_VEL
LIN {X 0,Y 576.421,Z 850.39,A -85,B 0,C 180,E1 9175.232,E2 9175.232} C_VEL
LIN {X 0,Y 575.203,Z 780.9,A -85,B 0,C 180,E1 9178.155,E2 9178.155} C_VEL
LIN {X 0,Y 570.64,Z 762.06,A -85,B 0,C 180,E1 9179.283,E2 9179.283} C_VEL
LIN {X 0,Y 570.553,Z 762.06,A -85,B 0,C 180,E1 9186.918,E2 9186.918} C_VEL
LIN {X 0,Y 570.353,Z 762.06,A -85,B 0,C 180,E1 9194.685,E2 9194.685} C_VEL
LIN {X 0,Y 569.97,Z 762.06,A -85,B 0,C 180,E1 9203.404,E2 9203.404} C_VEL
LIN {X 0,Y 569.961,Z 762.06,A -85,B 0,C 180,E1 9211.324,E2 9211.324} C_VEL
LIN {X 0,Y 570.061,Z 763.978,A -85,B 0,C 180,E1 9217.588,E2 9217.588} C_VEL
LIN {X 0,Y 610.949,Z 830.367,A -85,B 0,C 180,E1 9223.498,E2 9223.498} C_VEL
LIN {X 0,Y 615.617,Z 844.175,A -85,B 0,C 180,E1 9224.277,E2 9224.277} C_VEL
LIN {X 0,Y 608.232,Z 926.633,A -85,B 0,C 180,E1 9226.735,E2 9226.735} C_VEL
LIN {X 0,Y 602.144,Z 978.151,A -85,B 0,C 180,E1 9229.266,E2 9229.266} C_VEL
LIN {X 0,Y 591.065,Z 1008.549,A -85,B 0,C 180,E1 9230.673,E2 9230.673} C_VEL
LIN {X 0,Y 580.414,Z 1072.461,A -85,B 0,C 180,E1 9236.138,E2 9236.138} C_VEL
LIN {X 0,Y 571.482,Z 1126.704,A -85,B 0,C 180,E1 9242.896,E2 9242.896} C_VEL
LIN {X 0,Y 566.194,Z 1168.09,A -85,B 0,C 180,E1 9250.472,E2 9250.472} C_VEL
LIN {X 0,Y 563.633,Z 1195.407,A -85,B 0,C 180,E1 9258.393,E2 9258.393} C_VEL
LIN {X 0,Y 563.17,Z 1206.852,A -85,B 0,C 180,E1 9264.63,E2 9264.63} C_VEL
LIN {X 0,Y 563.061,Z 1209.864,A -85,B 0,C 180,E1 9270.813,E2 9270.813} C_VEL
LIN {X 0,Y 563.049,Z 1203.461,A -85,B 0,C 180,E1 9277.785,E2 9277.785} C_VEL
LIN {X 0,Y 563.976,Z 1186.044,A -85,B 0,C 180,E1 9284.851,E2 9284.851} C_VEL
LIN {X 0,Y 567.203,Z 1155.147,A -85,B 0,C 180,E1 9292.275,E2 9292.275} C_VEL
LIN {X 0,Y 574.081,Z 1109.577,A -85,B 0,C 180,E1 9299.536,E2 9299.536} C_VEL
LIN {X 0,Y 584.045,Z 1050.577,A -85,B 0,C 180,E1 9305.971,E2 9305.971} C_VEL
LIN {X 0,Y 594.762,Z 985.049,A -85,B 0,C 180,E1 9310.836,E2 9310.836} C_VEL
LIN {X 0,Y 604.167,Z 912.565,A -85,B 0,C 180,E1 9314.287,E2 9314.287} C_VEL
LIN {X 0,Y 608.826,Z 841.194,A -85,B 0,C 180,E1 9316.436,E2 9316.436} C_VEL
LIN {X 0,Y 573.443,Z 780.715,A -85,B 0,C 180,E1 9321.65,E2 9321.65} C_VEL
LIN {X 0,Y 562.163,Z 762.06,A -85,B 0,C 180,E1 9323.737,E2 9323.737} C_VEL
LIN {X 0,Y 562.383,Z 762.06,A -85,B 0,C 180,E1 9331.776,E2 9331.776} C_VEL
LIN {X 0,Y 562.084,Z 762.06,A -85,B 0,C 180,E1 9340.232,E2 9340.232} C_VEL
LIN {X 0,Y 562.612,Z 762.06,A -85,B 0,C 180,E1 9349.858,E2 9349.858} C_VEL
LIN {X 0,Y 563.449,Z 762.06,A -85,B 0,C 180,E1 9359.183,E2 9359.183} C_VEL
LIN {X 0,Y 562.634,Z 762.06,A -85,B 0,C 180,E1 9368.484,E2 9368.484} C_VEL
LIN {X 0,Y 562.24,Z 762.06,A -85,B 0,C 180,E1 9376.511,E2 9376.511} C_VEL
LIN {X 0,Y 562.175,Z 762.06,A -85,B 0,C 180,E1 9385.191,E2 9385.191} C_VEL
LIN {X 0,Y 561.927,Z 762.06,A -85,B 0,C 180,E1 9394.484,E2 9394.484} C_VEL
LIN {X 0,Y 562.132,Z 763.757,A -85,B 0,C 180,E1 9399.036,E2 9399.036} C_VEL
LIN {X 0,Y 583.744,Z 806.029,A -85,B 0,C 180,E1 9402.384,E2 9402.384} C_VEL
LIN {X 0,Y 605.025,Z 845.8,A -85,B 0,C 180,E1 9404.814,E2 9404.814} C_VEL
LIN {X 0,Y 598.57,Z 920.23,A -85,B 0,C 180,E1 9407.407,E2 9407.407} C_VEL
LIN {X 0,Y 590.132,Z 984.454,A -85,B 0,C 180,E1 9411.056,E2 9411.056} C_VEL
LIN {X 0,Y 579.042,Z 1048.896,A -85,B 0,C 180,E1 9416.755,E2 9416.755} C_VEL
LIN {X 0,Y 570.314,Z 1101.896,A -85,B 0,C 180,E1 9423.614,E2 9423.614} C_VEL
LIN {X 0,Y 565.558,Z 1137.86,A -85,B 0,C 180,E1 9430.362,E2 9430.362} C_VEL
LIN {X 0,Y 563.427,Z 1162.134,A -85,B 0,C 180,E1 9437.121,E2 9437.121} C_VEL
LIN {X 0,Y 562.988,Z 1175.818,A -85,B 0,C 180,E1 9443.77,E2 9443.77} C_VEL
LIN {X 0,Y 563.06,Z 1179.905,A -85,B 0,C 180,E1 9450.731,E2 9450.731} C_VEL
LIN {X 0,Y 563.498,Z 1172.091,A -85,B 0,C 180,E1 9458.475,E2 9458.475} C_VEL
LIN {X 0,Y 564.497,Z 1150.769,A -85,B 0,C 180,E1 9466.351,E2 9466.351} C_VEL
LIN {X 0,Y 568.289,Z 1116.713,A -85,B 0,C 180,E1 9473.791,E2 9473.791} C_VEL
LIN {X 0,Y 575.413,Z 1070.252,A -85,B 0,C 180,E1 9480.678,E2 9480.678} C_VEL
LIN {X 0,Y 585.858,Z 1009.695,A -85,B 0,C 180,E1 9486.872,E2 9486.872} C_VEL
LIN {X 0,Y 594.89,Z 950.573,A -85,B 0,C 180,E1 9490.989,E2 9490.989} C_VEL
LIN {X 0,Y 602.539,Z 875.357,A -85,B 0,C 180,E1 9494.263,E2 9494.263} C_VEL
LIN {X 0,Y 603.805,Z 838.976,A -85,B 0,C 180,E1 9495.374,E2 9495.374} C_VEL
LIN {X 0,Y 575.341,Z 787.399,A -85,B 0,C 180,E1 9498.775,E2 9498.775} C_VEL
LIN {X 0,Y 562.263,Z 762.06,A -85,B 0,C 180,E1 9500.983,E2 9500.983} C_VEL
LIN {X 0,Y 562.598,Z 763.586,A -85,B 0,C 180,E1 9502.558,E2 9502.558} C_VEL
LIN {X 0,Y 569.609,Z 806.272,A -85,B 0,C 180,E1 9504.647,E2 9504.647} C_VEL
LIN {X 0,Y 567.863,Z 860.369,A -85,B 0,C 180,E1 9506.75,E2 9506.75} C_VEL
LIN {X 0,Y 567.759,Z 987.861,A -85,B 0,C 180,E1 9508.702,E2 9508.702} C_VEL
LIN {X 0,Y 566.824,Z 1027.003,A -85,B 0,C 180,E1 9510.809,E2 9510.809} C_VEL
LIN {X 0,Y 565.6,Z 1056.84,A -85,B 0,C 180,E1 9514.089,E2 9514.089} C_VEL
LIN {X 0,Y 564.845,Z 1073.216,A -85,B 0,C 180,E1 9517.828,E2 9517.828} C_VEL
LIN {X 0,Y 564.865,Z 1076.808,A -85,B 0,C 180,E1 9522.342,E2 9522.342} C_VEL
LIN {X 0,Y 565.629,Z 1065.5,A -85,B 0,C 180,E1 9526.472,E2 9526.472} C_VEL
LIN {X 0,Y 566.418,Z 1040.716,A -85,B 0,C 180,E1 9530.019,E2 9530.019} C_VEL
LIN {X 0,Y 567.438,Z 1004.544,A -85,B 0,C 180,E1 9532.555,E2 9532.555} C_VEL
LIN {X 0,Y 567.61,Z 959.756,A -85,B 0,C 180,E1 9533.763,E2 9533.763} C_VEL
LIN {X 0,Y 568.714,Z 851.518,A -85,B 0,C 180,E1 9535.406,E2 9535.406} C_VEL
LIN {X 0,Y 567.41,Z 782.054,A -85,B 0,C 180,E1 9538.35,E2 9538.35} C_VEL
LIN {X 0,Y 562.594,Z 762.06,A -85,B 0,C 180,E1 9539.466,E2 9539.466} C_VEL
LIN {X 0,Y 562.521,Z 762.06,A -85,B 0,C 180,E1 9547.017,E2 9547.017} C_VEL
LIN {X 0,Y 562.297,Z 762.06,A -85,B 0,C 180,E1 9554.9,E2 9554.9} C_VEL
LIN {X 0,Y 561.998,Z 762.06,A -85,B 0,C 180,E1 9563.095,E2 9563.095} C_VEL
LIN {X 0,Y 561.892,Z 762.06,A -85,B 0,C 180,E1 9571.826,E2 9571.826} C_VEL
LIN {X 0,Y 562.027,Z 763.708,A -85,B 0,C 180,E1 9576.513,E2 9576.513} C_VEL
LIN {X 0,Y 604.694,Z 832.728,A -85,B 0,C 180,E1 9582.948,E2 9582.948} C_VEL
LIN {X 0,Y 609.698,Z 846.899,A -85,B 0,C 180,E1 9583.804,E2 9583.804} C_VEL
LIN {X 0,Y 601.937,Z 928.876,A -85,B 0,C 180,E1 9586.312,E2 9586.312} C_VEL
LIN {X 0,Y 592.225,Z 1001.323,A -85,B 0,C 180,E1 9590.19,E2 9590.19} C_VEL
LIN {X 0,Y 591.065,Z 1008.549,A -85,B 0,C 180,E1 9590.673,E2 9590.673} C_VEL
LIN {X 0,Y 579.624,Z 1037.323,A -85,B 0,C 180,E1 9592.377,E2 9592.377} C_VEL
LIN {X 0,Y 568.702,Z 1098.071,A -85,B 0,C 180,E1 9598.564,E2 9598.564} C_VEL
LIN {X 0,Y 560.506,Z 1147.118,A -85,B 0,C 180,E1 9605.875,E2 9605.875} C_VEL
LIN {X 0,Y 556.715,Z 1179.009,A -85,B 0,C 180,E1 9612.889,E2 9612.889} C_VEL
LIN {X 0,Y 555.223,Z 1199.092,A -85,B 0,C 180,E1 9619.81,E2 9619.81} C_VEL
LIN {X 0,Y 555.012,Z 1209.028,A -85,B 0,C 180,E1 9626.98,E2 9626.98} C_VEL
LIN {X 0,Y 555.207,Z 1208.317,A -85,B 0,C 180,E1 9633.959,E2 9633.959} C_VEL
LIN {X 0,Y 555.76,Z 1195.189,A -85,B 0,C 180,E1 9641.858,E2 9641.858} C_VEL
LIN {X 0,Y 557.662,Z 1169.489,A -85,B 0,C 180,E1 9649.514,E2 9649.514} C_VEL
LIN {X 0,Y 563.068,Z 1130.92,A -85,B 0,C 180,E1 9656.868,E2 9656.868} C_VEL
LIN {X 0,Y 572.478,Z 1076.845,A -85,B 0,C 180,E1 9663.868,E2 9663.868} C_VEL
LIN {X 0,Y 583.505,Z 1015.463,A -85,B 0,C 180,E1 9669.324,E2 9669.324} C_VEL
LIN {X 0,Y 593.916,Z 947.038,A -85,B 0,C 180,E1 9673.378,E2 9673.378} C_VEL
LIN {X 0,Y 602.416,Z 868.2,A -85,B 0,C 180,E1 9676.229,E2 9676.229} C_VEL
LIN {X 0,Y 602.987,Z 844.492,A -85,B 0,C 180,E1 9676.901,E2 9676.901} C_VEL
LIN {X 0,Y 568.502,Z 785.335,A -85,B 0,C 180,E1 9682.174,E2 9682.174} C_VEL
LIN {X 0,Y 554.167,Z 762.06,A -85,B 0,C 180,E1 9684.908,E2 9684.908} C_VEL
LIN {X 0,Y 554.399,Z 762.06,A -85,B 0,C 180,E1 9693.104,E2 9693.104} C_VEL
LIN {X 0,Y 554.349,Z 762.06,A -85,B 0,C 180,E1 9703.251,E2 9703.251} C_VEL
LIN {X 0,Y 554.635,Z 762.06,A -85,B 0,C 180,E1 9712.883,E2 9712.883} C_VEL
LIN {X 0,Y 554.796,Z 762.06,A -85,B 0,C 180,E1 9720.738,E2 9720.738} C_VEL
LIN {X 0,Y 554.594,Z 762.06,A -85,B 0,C 180,E1 9728.608,E2 9728.608} C_VEL
LIN {X 0,Y 554.224,Z 762.06,A -85,B 0,C 180,E1 9736.657,E2 9736.657} C_VEL
LIN {X 0,Y 554.182,Z 762.06,A -85,B 0,C 180,E1 9745.059,E2 9745.059} C_VEL
LIN {X 0,Y 553.916,Z 762.06,A -85,B 0,C 180,E1 9754.106,E2 9754.106} C_VEL
LIN {X 0,Y 554.204,Z 763.813,A -85,B 0,C 180,E1 9758.073,E2 9758.073} C_VEL
LIN {X 0,Y 576.17,Z 805.721,A -85,B 0,C 180,E1 9761.684,E2 9761.684} C_VEL
LIN {X 0,Y 598.027,Z 849.609,A -85,B 0,C 180,E1 9764.488,E2 9764.488} C_VEL
LIN {X 0,Y 590.942,Z 927.201,A -85,B 0,C 180,E1 9767.307,E2 9767.307} C_VEL
LIN {X 0,Y 581.62,Z 996.341,A -85,B 0,C 180,E1 9771.456,E2 9771.456} C_VEL
LIN {X 0,Y 570.363,Z 1058.265,A -85,B 0,C 180,E1 9777.356,E2 9777.356} C_VEL
LIN {X 0,Y 561.762,Z 1108.777,A -85,B 0,C 180,E1 9784.385,E2 9784.385} C_VEL
LIN {X 0,Y 557.176,Z 1144.631,A -85,B 0,C 180,E1 9791.706,E2 9791.706} C_VEL
LIN {X 0,Y 555.439,Z 1167.258,A -85,B 0,C 180,E1 9798.969,E2 9798.969} C_VEL
LIN {X 0,Y 555.31,Z 1178.346,A -85,B 0,C 180,E1 9806.041,E2 9806.041} C_VEL
LIN {X 0,Y 555.133,Z 1178.339,A -85,B 0,C 180,E1 9813.877,E2 9813.877} C_VEL
LIN {X 0,Y 555.247,Z 1167.346,A -85,B 0,C 180,E1 9820.907,E2 9820.907} C_VEL
LIN {X 0,Y 556.916,Z 1146.221,A -85,B 0,C 180,E1 9827.791,E2 9827.791} C_VEL
LIN {X 0,Y 561.29,Z 1111.313,A -85,B 0,C 180,E1 9835.107,E2 9835.107} C_VEL
LIN {X 0,Y 569.698,Z 1061.926,A -85,B 0,C 180,E1 9842.139,E2 9842.139} C_VEL
LIN {X 0,Y 580.999,Z 999.635,A -85,B 0,C 180,E1 9848.213,E2 9848.213} C_VEL
LIN {X 0,Y 590.578,Z 931.077,A -85,B 0,C 180,E1 9852.406,E2 9852.406} C_VEL
LIN {X 0,Y 597.736,Z 854.755,A -85,B 0,C 180,E1 9855.28,E2 9855.28} C_VEL
LIN {X 0,Y 596.296,Z 841.006,A -85,B 0,C 180,E1 9855.782,E2 9855.782} C_VEL
LIN {X 0,Y 569.444,Z 790.267,A -85,B 0,C 180,E1 9859.307,E2 9859.307} C_VEL
LIN {X 0,Y 554.421,Z 762.06,A -85,B 0,C 180,E1 9862.052,E2 9862.052} C_VEL
LIN {X 0,Y 561.914,Z 808.16,A -85,B 0,C 180,E1 9864.488,E2 9864.488} C_VEL
LIN {X 0,Y 560.114,Z 861.873,A -85,B 0,C 180,E1 9866.571,E2 9866.571} C_VEL
LIN {X 0,Y 559.962,Z 987.935,A -85,B 0,C 180,E1 9868.522,E2 9868.522} C_VEL
LIN {X 0,Y 559.002,Z 1027.353,A -85,B 0,C 180,E1 9870.633,E2 9870.633} C_VEL
LIN {X 0,Y 557.745,Z 1057.014,A -85,B 0,C 180,E1 9873.869,E2 9873.869} C_VEL
LIN {X 0,Y 556.951,Z 1074.76,A -85,B 0,C 180,E1 9877.985,E2 9877.985} C_VEL
LIN {X 0,Y 556.935,Z 1078.361,A -85,B 0,C 180,E1 9881.79,E2 9881.79} C_VEL
LIN {X 0,Y 557.536,Z 1069.408,A -85,B 0,C 180,E1 9885.87,E2 9885.87} C_VEL
LIN {X 0,Y 558.459,Z 1045.985,A -85,B 0,C 180,E1 9889.677,E2 9889.677} C_VEL
LIN {X 0,Y 559.641,Z 1011.684,A -85,B 0,C 180,E1 9892.389,E2 9892.389} C_VEL
LIN {X 0,Y 559.834,Z 971.206,A -85,B 0,C 180,E1 9893.773,E2 9893.773} C_VEL
LIN {X 0,Y 560.99,Z 852.792,A -85,B 0,C 180,E1 9895.586,E2 9895.586} C_VEL
LIN {X 0,Y 559.926,Z 784.488,A -85,B 0,C 180,E1 9898.493,E2 9898.493} C_VEL
LIN {X 0,Y 554.565,Z 762.06,A -85,B 0,C 180,E1 9899.654,E2 9899.654} C_VEL
LIN {X 0,Y 554.515,Z 762.06,A -85,B 0,C 180,E1 9907.119,E2 9907.119} C_VEL
LIN {X 0,Y 554.26,Z 762.06,A -85,B 0,C 180,E1 9915.121,E2 9915.121} C_VEL
LIN {X 0,Y 553.945,Z 762.06,A -85,B 0,C 180,E1 9923.525,E2 9923.525} C_VEL
LIN {X 0,Y 553.81,Z 762.06,A -85,B 0,C 180,E1 9932.346,E2 9932.346} C_VEL
LIN {X 0,Y 554.047,Z 763.912,A -85,B 0,C 180,E1 9935.404,E2 9935.404} C_VEL
LIN {X 0,Y 596.118,Z 830.815,A -85,B 0,C 180,E1 9942.041,E2 9942.041} C_VEL
LIN {X 0,Y 603.896,Z 849.054,A -85,B 0,C 180,E1 9943.31,E2 9943.31} C_VEL
LIN {X 0,Y 595.592,Z 932.086,A -85,B 0,C 180,E1 9945.917,E2 9945.917} C_VEL
LIN {X 0,Y 585.436,Z 1003.821,A -85,B 0,C 180,E1 9949.848,E2 9949.848} C_VEL
LIN {X 0,Y 579.624,Z 1037.323,A -85,B 0,C 180,E1 9952.377,E2 9952.377} C_VEL
LIN {X 0,Y 567.987,Z 1064.333,A -85,B 0,C 180,E1 9954.362,E2 9954.362} C_VEL
LIN {X 0,Y 557.592,Z 1119.644,A -85,B 0,C 180,E1 9961.026,E2 9961.026} C_VEL
LIN {X 0,Y 550.896,Z 1163.45,A -85,B 0,C 180,E1 9968.817,E2 9968.817} C_VEL
LIN {X 0,Y 548.145,Z 1193.357,A -85,B 0,C 180,E1 9977.249,E2 9977.249} C_VEL
LIN {X 0,Y 547.217,Z 1206.85,A -85,B 0,C 180,E1 9984.473,E2 9984.473} C_VEL
LIN {X 0,Y 547.056,Z 1209.864,A -85,B 0,C 180,E1 9990.837,E2 9990.837} C_VEL
LIN {X 0,Y 547.07,Z 1203.462,A -85,B 0,C 180,E1 9998.014,E2 9998.014} C_VEL
LIN {X 0,Y 548.206,Z 1186.043,A -85,B 0,C 180,E1 10005.288,E2 10005.288} C_VEL
LIN {X 0,Y 552.335,Z 1153.213,A -85,B 0,C 180,E1 10013.298,E2 10013.298} C_VEL
LIN {X 0,Y 560.042,Z 1107.258,A -85,B 0,C 180,E1 10020.682,E2 10020.682} C_VEL
LIN {X 0,Y 571.102,Z 1047.842,A -85,B 0,C 180,E1 10027.213,E2 10027.213} C_VEL
LIN {X 0,Y 582.939,Z 980.827,A -85,B 0,C 180,E1 10032.144,E2 10032.144} C_VEL
LIN {X 0,Y 593.096,Z 906.279,A -85,B 0,C 180,E1 10035.591,E2 10035.591} C_VEL
LIN {X 0,Y 597.161,Z 847.768,A -85,B 0,C 180,E1 10037.386,E2 10037.386} C_VEL
LIN {X 0,Y 561.91,Z 787.141,A -85,B 0,C 180,E1 10042.976,E2 10042.976} C_VEL
LIN {X 0,Y 546.168,Z 762.06,A -85,B 0,C 180,E1 10045.919,E2 10045.919} C_VEL
LIN {X 0,Y 546.375,Z 762.06,A -85,B 0,C 180,E1 10054.594,E2 10054.594} C_VEL
LIN {X 0,Y 546.302,Z 762.06,A -85,B 0,C 180,E1 10064.653,E2 10064.653} C_VEL
LIN {X 0,Y 546.633,Z 762.06,A -85,B 0,C 180,E1 10072.778,E2 10072.778} C_VEL
LIN {X 0,Y 546.801,Z 762.06,A -85,B 0,C 180,E1 10080.748,E2 10080.748} C_VEL
LIN {X 0,Y 546.409,Z 762.06,A -85,B 0,C 180,E1 10089.41,E2 10089.41} C_VEL
LIN {X 0,Y 546.024,Z 762.06,A -85,B 0,C 180,E1 10098.587,E2 10098.587} C_VEL
LIN {X 0,Y 546.096,Z 762.06,A -85,B 0,C 180,E1 10107.233,E2 10107.233} C_VEL
LIN {X 0,Y 545.925,Z 762.554,A -85,B 0,C 180,E1 10116.956,E2 10116.956} C_VEL
LIN {X 0,Y 569.754,Z 807.716,A -85,B 0,C 180,E1 10121.108,E2 10121.108} C_VEL
LIN {X 0,Y 591.068,Z 852.216,A -85,B 0,C 180,E1 10124.144,E2 10124.144} C_VEL
LIN {X 0,Y 583.646,Z 929.618,A -85,B 0,C 180,E1 10127.032,E2 10127.032} C_VEL
LIN {X 0,Y 574.68,Z 995.711,A -85,B 0,C 180,E1 10131.003,E2 10131.003} C_VEL
LIN {X 0,Y 564.875,Z 1049.85,A -85,B 0,C 180,E1 10135.933,E2 10135.933} C_VEL
LIN {X 0,Y 555.225,Z 1102.571,A -85,B 0,C 180,E1 10142.959,E2 10142.959} C_VEL
LIN {X 0,Y 549.781,Z 1139.61,A -85,B 0,C 180,E1 10150.195,E2 10150.195} C_VEL
LIN {X 0,Y 547.42,Z 1164.322,A -85,B 0,C 180,E1 10157.552,E2 10157.552} C_VEL
LIN {X 0,Y 547.089,Z 1176.847,A -85,B 0,C 180,E1 10164.387,E2 10164.387} C_VEL
LIN {X 0,Y 547.328,Z 1179.334,A -85,B 0,C 180,E1 10172.341,E2 10172.341} C_VEL
LIN {X 0,Y 547.3,Z 1169.025,A -85,B 0,C 180,E1 10180.339,E2 10180.339} C_VEL
LIN {X 0,Y 548.876,Z 1147.704,A -85,B 0,C 180,E1 10187.661,E2 10187.661} C_VEL
LIN {X 0,Y 553.237,Z 1114.594,A -85,B 0,C 180,E1 10194.895,E2 10194.895} C_VEL
LIN {X 0,Y 561.651,Z 1066.949,A -85,B 0,C 180,E1 10201.969,E2 10201.969} C_VEL
LIN {X 0,Y 572.294,Z 1010.114,A -85,B 0,C 180,E1 10207.794,E2 10207.794} C_VEL
LIN {X 0,Y 582.195,Z 942.749,A -85,B 0,C 180,E1 10212.225,E2 10212.225} C_VEL
LIN {X 0,Y 589.964,Z 864.768,A -85,B 0,C 180,E1 10215.408,E2 10215.408} C_VEL
LIN {X 0,Y 589.919,Z 845.208,A -85,B 0,C 180,E1 10216.05,E2 10216.05} C_VEL
LIN {X 0,Y 553.037,Z 774.405,A -85,B 0,C 180,E1 10221.646,E2 10221.646} C_VEL
LIN {X 0,Y 548.248,Z 770.856,A -85,B 0,C 180,E1 10222.382,E2 10222.382} C_VEL
LIN {X 0,Y 554.206,Z 809.879,A -85,B 0,C 180,E1 10224.316,E2 10224.316} C_VEL
LIN {X 0,Y 552.376,Z 865.189,A -85,B 0,C 180,E1 10226.417,E2 10226.417} C_VEL
LIN {X 0,Y 552.174,Z 989.767,A -85,B 0,C 180,E1 10228.391,E2 10228.391} C_VEL
LIN {X 0,Y 551.177,Z 1029.066,A -85,B 0,C 180,E1 10230.557,E2 10230.557} C_VEL
LIN {X 0,Y 549.852,Z 1058.906,A -85,B 0,C 180,E1 10233.912,E2 10233.912} C_VEL
LIN {X 0,Y 549.019,Z 1076.305,A -85,B 0,C 180,E1 10238.144,E2 10238.144} C_VEL
LIN {X 0,Y 549.036,Z 1079.106,A -85,B 0,C 180,E1 10242.311,E2 10242.311} C_VEL
LIN {X 0,Y 549.837,Z 1068.323,A -85,B 0,C 180,E1 10246.482,E2 10246.482} C_VEL
LIN {X 0,Y 550.701,Z 1043.989,A -85,B 0,C 180,E1 10250.132,E2 10250.132} C_VEL
LIN {X 0,Y 551.828,Z 1009.065,A -85,B 0,C 180,E1 10252.722,E2 10252.722} C_VEL
LIN {X 0,Y 552.01,Z 965.25,A -85,B 0,C 180,E1 10254.031,E2 10254.031} C_VEL
LIN {X 0,Y 553.272,Z 854.109,A -85,B 0,C 180,E1 10255.77,E2 10255.77} C_VEL
LIN {X 0,Y 552.259,Z 786.11,A -85,B 0,C 180,E1 10258.676,E2 10258.676} C_VEL
LIN {X 0,Y 546.518,Z 762.06,A -85,B 0,C 180,E1 10260.047,E2 10260.047} C_VEL
LIN {X 0,Y 546.487,Z 762.06,A -85,B 0,C 180,E1 10267.224,E2 10267.224} C_VEL
LIN {X 0,Y 546.21,Z 762.06,A -85,B 0,C 180,E1 10275.349,E2 10275.349} C_VEL
LIN {X 0,Y 545.922,Z 762.06,A -85,B 0,C 180,E1 10283.816,E2 10283.816} C_VEL
LIN {X 0,Y 545.794,Z 762.06,A -85,B 0,C 180,E1 10292.881,E2 10292.881} C_VEL
LIN {X 0,Y 546.11,Z 764.289,A -85,B 0,C 180,E1 10294.241,E2 10294.241} C_VEL
LIN {X 0,Y 587.077,Z 828.275,A -85,B 0,C 180,E1 10301.038,E2 10301.038} C_VEL
LIN {X 0,Y 597.943,Z 853.249,A -85,B 0,C 180,E1 10302.857,E2 10302.857} C_VEL
LIN {X 0,Y 589.243,Z 935.917,A -85,B 0,C 180,E1 10305.545,E2 10305.545} C_VEL
LIN {X 0,Y 578.551,Z 1007.082,A -85,B 0,C 180,E1 10309.541,E2 10309.541} C_VEL
LIN {X 0,Y 567.987,Z 1064.333,A -85,B 0,C 180,E1 10314.362,E2 10314.362} C_VEL
LIN {X 0,Y 556.237,Z 1089.485,A -85,B 0,C 180,E1 10316.625,E2 10316.625} C_VEL
LIN {X 0,Y 546.912,Z 1140.151,A -85,B 0,C 180,E1 10323.916,E2 10323.916} C_VEL
LIN {X 0,Y 541.23,Z 1178.011,A -85,B 0,C 180,E1 10332.098,E2 10332.098} C_VEL
LIN {X 0,Y 539.295,Z 1199.089,A -85,B 0,C 180,E1 10339.506,E2 10339.506} C_VEL
LIN {X 0,Y 538.942,Z 1208.385,A -85,B 0,C 180,E1 10346.007,E2 10346.007} C_VEL
LIN {X 0,Y 538.949,Z 1209.351,A -85,B 0,C 180,E1 10352.463,E2 10352.463} C_VEL
LIN {X 0,Y 539.632,Z 1199.895,A -85,B 0,C 180,E1 10360.105,E2 10360.105} C_VEL
LIN {X 0,Y 541.546,Z 1176.454,A -85,B 0,C 180,E1 10368.321,E2 10368.321} C_VEL
LIN {X 0,Y 546.97,Z 1138.381,A -85,B 0,C 180,E1 10376.397,E2 10376.397} C_VEL
LIN {X 0,Y 556.693,Z 1086.929,A -85,B 0,C 180,E1 10383.688,E2 10383.688} C_VEL
LIN {X 0,Y 568.729,Z 1026.521,A -85,B 0,C 180,E1 10389.55,E2 10389.55} C_VEL
LIN {X 0,Y 580.307,Z 958.815,A -85,B 0,C 180,E1 10393.915,E2 10393.915} C_VEL
LIN {X 0,Y 589.93,Z 879.615,A -85,B 0,C 180,E1 10397.024,E2 10397.024} C_VEL
LIN {X 0,Y 591.401,Z 851.29,A -85,B 0,C 180,E1 10397.851,E2 10397.851} C_VEL
LIN {X 0,Y 554.892,Z 788.131,A -85,B 0,C 180,E1 10403.892,E2 10403.892} C_VEL
LIN {X 0,Y 538.184,Z 762.06,A -85,B 0,C 180,E1 10407.245,E2 10407.245} C_VEL
LIN {X 0,Y 538.196,Z 762.06,A -85,B 0,C 180,E1 10416.494,E2 10416.494} C_VEL
LIN {X 0,Y 538.26,Z 762.06,A -85,B 0,C 180,E1 10426.088,E2 10426.088} C_VEL
LIN {X 0,Y 538.474,Z 762.06,A -85,B 0,C 180,E1 10434.293,E2 10434.293} C_VEL
LIN {X 0,Y 538.821,Z 762.06,A -85,B 0,C 180,E1 10440.759,E2 10440.759} C_VEL
LIN {X 0,Y 538.529,Z 762.06,A -85,B 0,C 180,E1 10448.866,E2 10448.866} C_VEL
LIN {X 0,Y 538.129,Z 762.06,A -85,B 0,C 180,E1 10457.171,E2 10457.171} C_VEL
LIN {X 0,Y 538.087,Z 762.06,A -85,B 0,C 180,E1 10465.863,E2 10465.863} C_VEL
LIN {X 0,Y 537.805,Z 762.06,A -85,B 0,C 180,E1 10475.437,E2 10475.437} C_VEL
LIN {X 0,Y 541.562,Z 768.922,A -85,B 0,C 180,E1 10476.579,E2 10476.579} C_VEL
LIN {X 0,Y 564.203,Z 811.358,A -85,B 0,C 180,E1 10480.643,E2 10480.643} C_VEL
LIN {X 0,Y 583.999,Z 854.946,A -85,B 0,C 180,E1 10483.805,E2 10483.805} C_VEL
LIN {X 0,Y 576.099,Z 934.281,A -85,B 0,C 180,E1 10486.862,E2 10486.862} C_VEL
LIN {X 0,Y 566.401,Z 1003.184,A -85,B 0,C 180,E1 10491.171,E2 10491.171} C_VEL
LIN {X 0,Y 556.774,Z 1055.751,A -85,B 0,C 180,E1 10496.134,E2 10496.134} C_VEL
LIN {X 0,Y 546.915,Z 1107.334,A -85,B 0,C 180,E1 10503.378,E2 10503.378} C_VEL
LIN {X 0,Y 541.561,Z 1143.069,A -85,B 0,C 180,E1 10510.734,E2 10510.734} C_VEL
LIN {X 0,Y 539.395,Z 1165.282,A -85,B 0,C 180,E1 10517.777,E2 10517.777} C_VEL
LIN {X 0,Y 539.1,Z 1176.846,A -85,B 0,C 180,E1 10524.304,E2 10524.304} C_VEL
LIN {X 0,Y 539.317,Z 1179.331,A -85,B 0,C 180,E1 10532.376,E2 10532.376} C_VEL
LIN {X 0,Y 539.328,Z 1169.026,A -85,B 0,C 180,E1 10540.493,E2 10540.493} C_VEL
LIN {X 0,Y 541.05,Z 1147.706,A -85,B 0,C 180,E1 10547.925,E2 10547.925} C_VEL
LIN {X 0,Y 545.911,Z 1113.249,A -85,B 0,C 180,E1 10555.517,E2 10555.517} C_VEL
LIN {X 0,Y 555.211,Z 1063.644,A -85,B 0,C 180,E1 10562.85,E2 10562.85} C_VEL
LIN {X 0,Y 564.956,Z 1011.5,A -85,B 0,C 180,E1 10568.084,E2 10568.084} C_VEL
LIN {X 0,Y 574.786,Z 945.606,A -85,B 0,C 180,E1 10572.467,E2 10572.467} C_VEL
LIN {X 0,Y 582.64,Z 869.224,A -85,B 0,C 180,E1 10575.682,E2 10575.682} C_VEL
LIN {X 0,Y 582.906,Z 848.306,A -85,B 0,C 180,E1 10576.382,E2 10576.382} C_VEL
LIN {X 0,Y 548.95,Z 780.691,A -85,B 0,C 180,E1 10581.956,E2 10581.956} C_VEL
LIN {X 0,Y 543.233,Z 784.061,A -85,B 0,C 180,E1 10582.799,E2 10582.799} C_VEL
LIN {X 0,Y 546.399,Z 818.163,A -85,B 0,C 180,E1 10584.426,E2 10584.426} C_VEL
LIN {X 0,Y 544.632,Z 865.449,A -85,B 0,C 180,E1 10586.212,E2 10586.212} C_VEL
LIN {X 0,Y 544.318,Z 991.357,A -85,B 0,C 180,E1 10588.249,E2 10588.249} C_VEL
LIN {X 0,Y 543.329,Z 1031.172,A -85,B 0,C 180,E1 10590.509,E2 10590.509} C_VEL
LIN {X 0,Y 541.989,Z 1060.021,A -85,B 0,C 180,E1 10593.835,E2 10593.835} C_VEL
LIN {X 0,Y 541.104,Z 1076.684,A -85,B 0,C 180,E1 10597.808,E2 10597.808} C_VEL
LIN {X 0,Y 541.082,Z 1080.732,A -85,B 0,C 180,E1 10601.237,E2 10601.237} C_VEL
LIN {X 0,Y 541.678,Z 1072.986,A -85,B 0,C 180,E1 10605.661,E2 10605.661} C_VEL
LIN {X 0,Y 542.778,Z 1051.015,A -85,B 0,C 180,E1 10609.579,E2 10609.579} C_VEL
LIN {X 0,Y 544.007,Z 1016.864,A -85,B 0,C 180,E1 10612.51,E2 10612.51} C_VEL
LIN {X 0,Y 544.246,Z 975.675,A -85,B 0,C 180,E1 10614.046,E2 10614.046} C_VEL
LIN {X 0,Y 545.589,Z 854.139,A -85,B 0,C 180,E1 10616.01,E2 10616.01} C_VEL
LIN {X 0,Y 544.398,Z 786.912,A -85,B 0,C 180,E1 10618.915,E2 10618.915} C_VEL
LIN {X 0,Y 538.52,Z 762.06,A -85,B 0,C 180,E1 10620.319,E2 10620.319} C_VEL
LIN {X 0,Y 538.459,Z 762.06,A -85,B 0,C 180,E1 10627.332,E2 10627.332} C_VEL
LIN {X 0,Y 538.184,Z 762.06,A -85,B 0,C 180,E1 10635.584,E2 10635.584} C_VEL
LIN {X 0,Y 537.89,Z 762.06,A -85,B 0,C 180,E1 10644.194,E2 10644.194} C_VEL
LIN {X 0,Y 537.967,Z 763.727,A -85,B 0,C 180,E1 10652.971,E2 10652.971} C_VEL
LIN {X 0,Y 579.378,Z 828.358,A -85,B 0,C 180,E1 10660.213,E2 10660.213} C_VEL
LIN {X 0,Y 592.202,Z 854.915,A -85,B 0,C 180,E1 10662.342,E2 10662.342} C_VEL
LIN {X 0,Y 583.19,Z 937.855,A -85,B 0,C 180,E1 10665.068,E2 10665.068} C_VEL
LIN {X 0,Y 571.85,Z 1010.029,A -85,B 0,C 180,E1 10669.196,E2 10669.196} C_VEL
LIN {X 0,Y 559.795,Z 1071.919,A -85,B 0,C 180,E1 10674.644,E2 10674.644} C_VEL
LIN {X 0,Y 556.237,Z 1089.485,A -85,B 0,C 180,E1 10676.625,E2 10676.625} C_VEL
LIN {X 0,Y 544.272,Z 1112.586,A -85,B 0,C 180,E1 10679.143,E2 10679.143} C_VEL
LIN {X 0,Y 536.043,Z 1157.495,A -85,B 0,C 180,E1 10686.861,E2 10686.861} C_VEL
LIN {X 0,Y 532.247,Z 1187.63,A -85,B 0,C 180,E1 10694.755,E2 10694.755} C_VEL
LIN {X 0,Y 531.414,Z 1204.799,A -85,B 0,C 180,E1 10702.662,E2 10702.662} C_VEL
LIN {X 0,Y 531.061,Z 1209.864,A -85,B 0,C 180,E1 10710.862,E2 10710.862} C_VEL
LIN {X 0,Y 531.14,Z 1203.459,A -85,B 0,C 180,E1 10718.256,E2 10718.256} C_VEL
LIN {X 0,Y 532.768,Z 1184.725,A -85,B 0,C 180,E1 10726.167,E2 10726.167} C_VEL
LIN {X 0,Y 537.765,Z 1150.363,A -85,B 0,C 180,E1 10734.563,E2 10734.563} C_VEL
LIN {X 0,Y 546.557,Z 1102.813,A -85,B 0,C 180,E1 10742.172,E2 10742.172} C_VEL
LIN {X 0,Y 558.86,Z 1044.745,A -85,B 0,C 180,E1 10748.568,E2 10748.568} C_VEL
LIN {X 0,Y 571.152,Z 979.675,A -85,B 0,C 180,E1 10753.348,E2 10753.348} C_VEL
LIN {X 0,Y 581.59,Z 906.745,A -85,B 0,C 180,E1 10756.688,E2 10756.688} C_VEL
LIN {X 0,Y 585.471,Z 854.445,A -85,B 0,C 180,E1 10758.347,E2 10758.347} C_VEL
LIN {X 0,Y 549.76,Z 792.718,A -85,B 0,C 180,E1 10764.463,E2 10764.463} C_VEL
LIN {X 0,Y 530.217,Z 762.06,A -85,B 0,C 180,E1 10768.427,E2 10768.427} C_VEL
LIN {X 0,Y 530.107,Z 762.06,A -85,B 0,C 180,E1 10777.218,E2 10777.218} C_VEL
LIN {X 0,Y 530.241,Z 762.06,A -85,B 0,C 180,E1 10785.874,E2 10785.874} C_VEL
LIN {X 0,Y 530.474,Z 762.06,A -85,B 0,C 180,E1 10794.206,E2 10794.206} C_VEL
LIN {X 0,Y 530.814,Z 762.06,A -85,B 0,C 180,E1 10800.771,E2 10800.771} C_VEL
LIN {X 0,Y 530.505,Z 762.06,A -85,B 0,C 180,E1 10809.062,E2 10809.062} C_VEL
LIN {X 0,Y 530.076,Z 762.06,A -85,B 0,C 180,E1 10817.44,E2 10817.44} C_VEL
LIN {X 0,Y 530.057,Z 762.06,A -85,B 0,C 180,E1 10826.285,E2 10826.285} C_VEL
LIN {X 0,Y 529.968,Z 763.833,A -85,B 0,C 180,E1 10834.707,E2 10834.707} C_VEL
LIN {X 0,Y 556.417,Z 809.33,A -85,B 0,C 180,E1 10839.729,E2 10839.729} C_VEL
LIN {X 0,Y 577.098,Z 856.799,A -85,B 0,C 180,E1 10843.416,E2 10843.416} C_VEL
LIN {X 0,Y 568.118,Z 941.167,A -85,B 0,C 180,E1 10846.81,E2 10846.81} C_VEL
LIN {X 0,Y 558.198,Z 1010.048,A -85,B 0,C 180,E1 10851.305,E2 10851.305} C_VEL
LIN {X 0,Y 547.805,Z 1065.806,A -85,B 0,C 180,E1 10856.868,E2 10856.868} C_VEL
LIN {X 0,Y 538.299,Z 1114.286,A -85,B 0,C 180,E1 10864.211,E2 10864.211} C_VEL
LIN {X 0,Y 533.251,Z 1149.601,A -85,B 0,C 180,E1 10872.239,E2 10872.239} C_VEL
LIN {X 0,Y 531.6,Z 1170.996,A -85,B 0,C 180,E1 10880.318,E2 10880.318} C_VEL
LIN {X 0,Y 531.09,Z 1179.33,A -85,B 0,C 180,E1 10887.5,E2 10887.5} C_VEL
LIN {X 0,Y 531.12,Z 1178.332,A -85,B 0,C 180,E1 10894.052,E2 10894.052} C_VEL
LIN {X 0,Y 531.369,Z 1167.156,A -85,B 0,C 180,E1 10901.486,E2 10901.486} C_VEL
LIN {X 0,Y 533.614,Z 1144.626,A -85,B 0,C 180,E1 10909.041,E2 10909.041} C_VEL
LIN {X 0,Y 539.839,Z 1106.131,A -85,B 0,C 180,E1 10917.129,E2 10917.129} C_VEL
LIN {X 0,Y 549.834,Z 1055.747,A -85,B 0,C 180,E1 10924.239,E2 10924.239} C_VEL
LIN {X 0,Y 560.377,Z 995.933,A -85,B 0,C 180,E1 10929.69,E2 10929.69} C_VEL
LIN {X 0,Y 570.215,Z 926.234,A -85,B 0,C 180,E1 10933.828,E2 10933.828} C_VEL
LIN {X 0,Y 576.334,Z 852.007,A -85,B 0,C 180,E1 10936.727,E2 10936.727} C_VEL
LIN {X 0,Y 546.365,Z 790.748,A -85,B 0,C 180,E1 10941.955,E2 10941.955} C_VEL
LIN {X 0,Y 537.538,Z 794.411,A -85,B 0,C 180,E1 10942.98,E2 10942.98} C_VEL
LIN {X 0,Y 537.364,Z 852.056,A -85,B 0,C 180,E1 10945.64,E2 10945.64} C_VEL
LIN {X 0,Y 536.528,Z 993.311,A -85,B 0,C 180,E1 10948.123,E2 10948.123} C_VEL
LIN {X 0,Y 535.481,Z 1032.99,A -85,B 0,C 180,E1 10950.445,E2 10950.445} C_VEL
LIN {X 0,Y 534.082,Z 1062.226,A -85,B 0,C 180,E1 10953.928,E2 10953.928} C_VEL
LIN {X 0,Y 533.218,Z 1077.203,A -85,B 0,C 180,E1 10957.529,E2 10957.529} C_VEL
LIN {X 0,Y 533.223,Z 1081.416,A -85,B 0,C 180,E1 10962.273,E2 10962.273} C_VEL
LIN {X 0,Y 534.031,Z 1071.11,A -85,B 0,C 180,E1 10966.493,E2 10966.493} C_VEL
LIN {X 0,Y 535.011,Z 1047.269,A -85,B 0,C 180,E1 10970.252,E2 10970.252} C_VEL
LIN {X 0,Y 536.26,Z 1012.901,A -85,B 0,C 180,E1 10972.937,E2 10972.937} C_VEL
LIN {X 0,Y 536.385,Z 971.062,A -85,B 0,C 180,E1 10974.315,E2 10974.315} C_VEL
LIN {X 0,Y 537.913,Z 855.548,A -85,B 0,C 180,E1 10976.206,E2 10976.206} C_VEL
LIN {X 0,Y 537.085,Z 789.939,A -85,B 0,C 180,E1 10979.042,E2 10979.042} C_VEL
LIN {X 0,Y 530.485,Z 762.06,A -85,B 0,C 180,E1 10980.505,E2 10980.505} C_VEL
LIN {X 0,Y 530.435,Z 762.06,A -85,B 0,C 180,E1 10987.444,E2 10987.444} C_VEL
LIN {X 0,Y 530.067,Z 762.06,A -85,B 0,C 180,E1 10996.627,E2 10996.627} C_VEL
LIN {X 0,Y 529.873,Z 762.06,A -85,B 0,C 180,E1 11006.402,E2 11006.402} C_VEL
LIN {X 0,Y 530.045,Z 764,A -85,B 0,C 180,E1 11011.679,E2 11011.679} C_VEL
LIN {X 0,Y 568.771,Z 823.795,A -85,B 0,C 180,E1 11018.878,E2 11018.878} C_VEL
LIN {X 0,Y 586.281,Z 859.31,A -85,B 0,C 180,E1 11021.893,E2 11021.893} C_VEL
LIN {X 0,Y 576.658,Z 943.647,A -85,B 0,C 180,E1 11024.763,E2 11024.763} C_VEL
LIN {X 0,Y 565.333,Z 1012.117,A -85,B 0,C 180,E1 11028.781,E2 11028.781} C_VEL
LIN {X 0,Y 553.086,Z 1071.842,A -85,B 0,C 180,E1 11034.102,E2 11034.102} C_VEL
LIN {X 0,Y 544.272,Z 1112.586,A -85,B 0,C 180,E1 11039.143,E2 11039.143} C_VEL
LIN {X 0,Y 533.156,Z 1133.477,A -85,B 0,C 180,E1 11041.962,E2 11041.962} C_VEL
LIN {X 0,Y 526.663,Z 1172.572,A -85,B 0,C 180,E1 11050.09,E2 11050.09} C_VEL
LIN {X 0,Y 523.716,Z 1197.32,A -85,B 0,C 180,E1 11058.344,E2 11058.344} C_VEL
LIN {X 0,Y 522.974,Z 1208.381,A -85,B 0,C 180,E1 11065.885,E2 11065.885} C_VEL
LIN {X 0,Y 522.961,Z 1209.348,A -85,B 0,C 180,E1 11072.539,E2 11072.539} C_VEL
LIN {X 0,Y 523.694,Z 1199.964,A -85,B 0,C 180,E1 11080.382,E2 11080.382} C_VEL
LIN {X 0,Y 525.786,Z 1176.1,A -85,B 0,C 180,E1 11088.991,E2 11088.991} C_VEL
LIN {X 0,Y 531.925,Z 1138.643,A -85,B 0,C 180,E1 11097.155,E2 11097.155} C_VEL
LIN {X 0,Y 543.433,Z 1084.863,A -85,B 0,C 180,E1 11104.969,E2 11104.969} C_VEL
LIN {X 0,Y 556.922,Z 1025.031,A -85,B 0,C 180,E1 11110.852,E2 11110.852} C_VEL
LIN {X 0,Y 568.686,Z 959.234,A -85,B 0,C 180,E1 11115.053,E2 11115.053} C_VEL
LIN {X 0,Y 578.955,Z 875.704,A -85,B 0,C 180,E1 11118.249,E2 11118.249} C_VEL
LIN {X 0,Y 579.373,Z 857.774,A -85,B 0,C 180,E1 11118.864,E2 11118.864} C_VEL
LIN {X 0,Y 545.581,Z 798.363,A -85,B 0,C 180,E1 11124.884,E2 11124.884} C_VEL
LIN {X 0,Y 522.239,Z 762.06,A -85,B 0,C 180,E1 11129.888,E2 11129.888} C_VEL
LIN {X 0,Y 522.018,Z 762.06,A -85,B 0,C 180,E1 11138.644,E2 11138.644} C_VEL
LIN {X 0,Y 522.22,Z 762.06,A -85,B 0,C 180,E1 11147.364,E2 11147.364} C_VEL
LIN {X 0,Y 522.46,Z 762.06,A -85,B 0,C 180,E1 11155.788,E2 11155.788} C_VEL
LIN {X 0,Y 522.529,Z 762.06,A -85,B 0,C 180,E1 11162.447,E2 11162.447} C_VEL
LIN {X 0,Y 522.313,Z 762.06,A -85,B 0,C 180,E1 11170.834,E2 11170.834} C_VEL
LIN {X 0,Y 522.002,Z 762.06,A -85,B 0,C 180,E1 11179.476,E2 11179.476} C_VEL
LIN {X 0,Y 521.976,Z 762.06,A -85,B 0,C 180,E1 11188.604,E2 11188.604} C_VEL
LIN {X 0,Y 521.967,Z 763.805,A -85,B 0,C 180,E1 11193.436,E2 11193.436} C_VEL
LIN {X 0,Y 550.382,Z 811.348,A -85,B 0,C 180,E1 11199.098,E2 11199.098} C_VEL
LIN {X 0,Y 570.429,Z 861.315,A -85,B 0,C 180,E1 11203.046,E2 11203.046} C_VEL
LIN {X 0,Y 559.541,Z 951.593,A -85,B 0,C 180,E1 11206.993,E2 11206.993} C_VEL
LIN {X 0,Y 549.665,Z 1017.332,A -85,B 0,C 180,E1 11211.549,E2 11211.549} C_VEL
LIN {X 0,Y 539.06,Z 1073.965,A -85,B 0,C 180,E1 11217.465,E2 11217.465} C_VEL
LIN {X 0,Y 529.756,Z 1120.775,A -85,B 0,C 180,E1 11225.098,E2 11225.098} C_VEL
LIN {X 0,Y 525.084,Z 1154.811,A -85,B 0,C 180,E1 11233.59,E2 11233.59} C_VEL
LIN {X 0,Y 523.375,Z 1173.539,A -85,B 0,C 180,E1 11241.621,E2 11241.621} C_VEL
LIN {X 0,Y 522.79,Z 1179.903,A -85,B 0,C 180,E1 11249.124,E2 11249.124} C_VEL
LIN {X 0,Y 523.207,Z 1175.798,A -85,B 0,C 180,E1 11256.617,E2 11256.617} C_VEL
LIN {X 0,Y 524.7,Z 1158.476,A -85,B 0,C 180,E1 11265.122,E2 11265.122} C_VEL
LIN {X 0,Y 528.806,Z 1126.321,A -85,B 0,C 180,E1 11273.675,E2 11273.675} C_VEL
LIN {X 0,Y 537.484,Z 1081.329,A -85,B 0,C 180,E1 11281.434,E2 11281.434} C_VEL
LIN {X 0,Y 548.083,Z 1026.667,A -85,B 0,C 180,E1 11287.559,E2 11287.559} C_VEL
LIN {X 0,Y 558.334,Z 961.611,A -85,B 0,C 180,E1 11292.347,E2 11292.347} C_VEL
LIN {X 0,Y 568.966,Z 874.152,A -85,B 0,C 180,E1 11296.428,E2 11296.428} C_VEL
LIN {X 0,Y 569.556,Z 854.728,A -85,B 0,C 180,E1 11297.213,E2 11297.213} C_VEL
LIN {X 0,Y 543.93,Z 800.214,A -85,B 0,C 180,E1 11301.951,E2 11301.951} C_VEL
LIN {X 0,Y 531.682,Z 807.11,A -85,B 0,C 180,E1 11303.32,E2 11303.32} C_VEL
LIN {X 0,Y 529.177,Z 863.921,A -85,B 0,C 180,E1 11305.755,E2 11305.755} C_VEL
LIN {X 0,Y 528.729,Z 992.414,A -85,B 0,C 180,E1 11307.887,E2 11307.887} C_VEL
LIN {X 0,Y 527.694,Z 1032.137,A -85,B 0,C 180,E1 11310.155,E2 11310.155} C_VEL
LIN {X 0,Y 526.252,Z 1061.239,A -85,B 0,C 180,E1 11313.51,E2 11313.51} C_VEL
LIN {X 0,Y 525.29,Z 1078.536,A -85,B 0,C 180,E1 11317.595,E2 11317.595} C_VEL
LIN {X 0,Y 525.259,Z 1082.883,A -85,B 0,C 180,E1 11321.525,E2 11321.525} C_VEL
LIN {X 0,Y 525.914,Z 1074.978,A -85,B 0,C 180,E1 11325.855,E2 11325.855} C_VEL
LIN {X 0,Y 527.099,Z 1052.573,A -85,B 0,C 180,E1 11329.894,E2 11329.894} C_VEL
LIN {X 0,Y 528.425,Z 1018.804,A -85,B 0,C 180,E1 11332.832,E2 11332.832} C_VEL
LIN {X 0,Y 528.648,Z 978.029,A -85,B 0,C 180,E1 11334.387,E2 11334.387} C_VEL
LIN {X 0,Y 530.221,Z 856.293,A -85,B 0,C 180,E1 11336.429,E2 11336.429} C_VEL
LIN {X 0,Y 529.566,Z 792.098,A -85,B 0,C 180,E1 11339.227,E2 11339.227} C_VEL
LIN {X 0,Y 522.529,Z 762.06,A -85,B 0,C 180,E1 11340.881,E2 11340.881} C_VEL
LIN {X 0,Y 522.31,Z 762.06,A -85,B 0,C 180,E1 11349.243,E2 11349.243} C_VEL
LIN {X 0,Y 522.026,Z 762.06,A -85,B 0,C 180,E1 11357.82,E2 11357.82} C_VEL
LIN {X 0,Y 521.805,Z 762.06,A -85,B 0,C 180,E1 11367.61,E2 11367.61} C_VEL
LIN {X 0,Y 522.039,Z 763.775,A -85,B 0,C 180,E1 11370.283,E2 11370.283} C_VEL
LIN {X 0,Y 560.627,Z 823.016,A -85,B 0,C 180,E1 11377.876,E2 11377.876} C_VEL
LIN {X 0,Y 580.517,Z 861.535,A -85,B 0,C 180,E1 11381.387,E2 11381.387} C_VEL
LIN {X 0,Y 570.363,Z 947.192,A -85,B 0,C 180,E1 11384.362,E2 11384.362} C_VEL
LIN {X 0,Y 558.969,Z 1014.904,A -85,B 0,C 180,E1 11388.368,E2 11388.368} C_VEL
LIN {X 0,Y 546.003,Z 1073.951,A -85,B 0,C 180,E1 11393.782,E2 11393.782} C_VEL
LIN {X 0,Y 533.991,Z 1128.729,A -85,B 0,C 180,E1 11401.164,E2 11401.164} C_VEL
LIN {X 0,Y 533.156,Z 1133.477,A -85,B 0,C 180,E1 11401.962,E2 11401.962} C_VEL
LIN {X 0,Y 521.72,Z 1152.13,A -85,B 0,C 180,E1 11405.014,E2 11405.014} C_VEL
LIN {X 0,Y 516.996,Z 1182.775,A -85,B 0,C 180,E1 11412.679,E2 11412.679} C_VEL
LIN {X 0,Y 515.265,Z 1200.719,A -85,B 0,C 180,E1 11419.869,E2 11419.869} C_VEL
LIN {X 0,Y 515.144,Z 1209.39,A -85,B 0,C 180,E1 11427.513,E2 11427.513} C_VEL
LIN {X 0,Y 515.244,Z 1206.746,A -85,B 0,C 180,E1 11435.961,E2 11435.961} C_VEL
LIN {X 0,Y 515.863,Z 1192.636,A -85,B 0,C 180,E1 11443.867,E2 11443.867} C_VEL
LIN {X 0,Y 518.962,Z 1167.714,A -85,B 0,C 180,E1 11451.484,E2 11451.484} C_VEL
LIN {X 0,Y 526.583,Z 1128.149,A -85,B 0,C 180,E1 11459.381,E2 11459.381} C_VEL
LIN {X 0,Y 539.897,Z 1072.642,A -85,B 0,C 180,E1 11466.977,E2 11466.977} C_VEL
LIN {X 0,Y 553.269,Z 1014.644,A -85,B 0,C 180,E1 11472.271,E2 11472.271} C_VEL
LIN {X 0,Y 564.508,Z 948.279,A -85,B 0,C 180,E1 11476.12,E2 11476.12} C_VEL
LIN {X 0,Y 573.469,Z 861.655,A -85,B 0,C 180,E1 11479.341,E2 11479.341} C_VEL
LIN {X 0,Y 542.004,Z 804.978,A -85,B 0,C 180,E1 11485.167,E2 11485.167} C_VEL
LIN {X 0,Y 514.225,Z 762.06,A -85,B 0,C 180,E1 11491.421,E2 11491.421} C_VEL
LIN {X 0,Y 514.017,Z 762.06,A -85,B 0,C 180,E1 11500.104,E2 11500.104} C_VEL
LIN {X 0,Y 514.389,Z 762.06,A -85,B 0,C 180,E1 11508.896,E2 11508.896} C_VEL
LIN {X 0,Y 515.411,Z 762.06,A -85,B 0,C 180,E1 11519.107,E2 11519.107} C_VEL
LIN {X 0,Y 514.49,Z 762.06,A -85,B 0,C 180,E1 11529.284,E2 11529.284} C_VEL
LIN {X 0,Y 514.016,Z 762.06,A -85,B 0,C 180,E1 11538.003,E2 11538.003} C_VEL
LIN {X 0,Y 513.984,Z 762.06,A -85,B 0,C 180,E1 11547.173,E2 11547.173} C_VEL
LIN {X 0,Y 514.099,Z 764.068,A -85,B 0,C 180,E1 11552.107,E2 11552.107} C_VEL
LIN {X 0,Y 542.908,Z 811.369,A -85,B 0,C 180,E1 11558.198,E2 11558.198} C_VEL
LIN {X 0,Y 564.179,Z 863.583,A -85,B 0,C 180,E1 11562.569,E2 11562.569} C_VEL
LIN {X 0,Y 552.753,Z 949.564,A -85,B 0,C 180,E1 11566.492,E2 11566.492} C_VEL
LIN {X 0,Y 542.265,Z 1018.041,A -85,B 0,C 180,E1 11571.235,E2 11571.235} C_VEL
LIN {X 0,Y 531.577,Z 1074.336,A -85,B 0,C 180,E1 11577.147,E2 11577.147} C_VEL
LIN {X 0,Y 522.527,Z 1118.176,A -85,B 0,C 180,E1 11584.189,E2 11584.189} C_VEL
LIN {X 0,Y 517.283,Z 1152.606,A -85,B 0,C 180,E1 11592.613,E2 11592.613} C_VEL
LIN {X 0,Y 515.411,Z 1173.539,A -85,B 0,C 180,E1 11601.49,E2 11601.49} C_VEL
LIN {X 0,Y 514.792,Z 1179.9,A -85,B 0,C 180,E1 11609.111,E2 11609.111} C_VEL
LIN {X 0,Y 515.253,Z 1175.796,A -85,B 0,C 180,E1 11616.72,E2 11616.72} C_VEL
LIN {X 0,Y 516.733,Z 1158.692,A -85,B 0,C 180,E1 11625.278,E2 11625.278} C_VEL
LIN {X 0,Y 520.962,Z 1127.524,A -85,B 0,C 180,E1 11633.777,E2 11633.777} C_VEL
LIN {X 0,Y 529.578,Z 1084.304,A -85,B 0,C 180,E1 11641.416,E2 11641.416} C_VEL
LIN {X 0,Y 539.655,Z 1032.822,A -85,B 0,C 180,E1 11647.344,E2 11647.344} C_VEL
LIN {X 0,Y 550.069,Z 969.114,A -85,B 0,C 180,E1 11652.259,E2 11652.259} C_VEL
LIN {X 0,Y 562.41,Z 878.504,A -85,B 0,C 180,E1 11656.813,E2 11656.813} C_VEL
LIN {X 0,Y 563.256,Z 858.327,A -85,B 0,C 180,E1 11657.66,E2 11657.66} C_VEL
LIN {X 0,Y 541.152,Z 809.939,A -85,B 0,C 180,E1 11661.975,E2 11661.975} C_VEL
LIN {X 0,Y 530.603,Z 819.228,A -85,B 0,C 180,E1 11663.027,E2 11663.027} C_VEL
LIN {X 0,Y 523.817,Z 824.242,A -85,B 0,C 180,E1 11663.774,E2 11663.774} C_VEL
LIN {X 0,Y 521.446,Z 868.743,A -85,B 0,C 180,E1 11665.605,E2 11665.605} C_VEL
LIN {X 0,Y 520.955,Z 993.04,A -85,B 0,C 180,E1 11667.703,E2 11667.703} C_VEL
LIN {X 0,Y 519.878,Z 1032.364,A -85,B 0,C 180,E1 11669.95,E2 11669.95} C_VEL
LIN {X 0,Y 518.357,Z 1063.249,A -85,B 0,C 180,E1 11673.569,E2 11673.569} C_VEL
LIN {X 0,Y 517.36,Z 1080.549,A -85,B 0,C 180,E1 11677.959,E2 11677.959} C_VEL
LIN {X 0,Y 517.421,Z 1083.727,A -85,B 0,C 180,E1 11682.229,E2 11682.229} C_VEL
LIN {X 0,Y 518.2,Z 1073.917,A -85,B 0,C 180,E1 11686.504,E2 11686.504} C_VEL
LIN {X 0,Y 519.332,Z 1050.599,A -85,B 0,C 180,E1 11690.379,E2 11690.379} C_VEL
LIN {X 0,Y 520.694,Z 1015.26,A -85,B 0,C 180,E1 11693.251,E2 11693.251} C_VEL
LIN {X 0,Y 520.847,Z 973.278,A -85,B 0,C 180,E1 11694.669,E2 11694.669} C_VEL
LIN {X 0,Y 522.491,Z 858.344,A -85,B 0,C 180,E1 11696.615,E2 11696.615} C_VEL
LIN {X 0,Y 521.566,Z 792.033,A -85,B 0,C 180,E1 11699.53,E2 11699.53} C_VEL
LIN {X 0,Y 514.543,Z 762.06,A -85,B 0,C 180,E1 11701.317,E2 11701.317} C_VEL
LIN {X 0,Y 514.324,Z 762.06,A -85,B 0,C 180,E1 11709.388,E2 11709.388} C_VEL
LIN {X 0,Y 514.012,Z 762.06,A -85,B 0,C 180,E1 11718.108,E2 11718.108} C_VEL
LIN {X 0,Y 513.796,Z 762.06,A -85,B 0,C 180,E1 11728.078,E2 11728.078} C_VEL
LIN {X 0,Y 514.351,Z 764.834,A -85,B 0,C 180,E1 11728.897,E2 11728.897} C_VEL
LIN {X 0,Y 550.226,Z 818.595,A -85,B 0,C 180,E1 11736.418,E2 11736.418} C_VEL
LIN {X 0,Y 574.674,Z 864.795,A -85,B 0,C 180,E1 11740.897,E2 11740.897} C_VEL
LIN {X 0,Y 563.999,Z 950.422,A -85,B 0,C 180,E1 11743.959,E2 11743.959} C_VEL
LIN {X 0,Y 552.66,Z 1017.535,A -85,B 0,C 180,E1 11747.935,E2 11747.935} C_VEL
LIN {X 0,Y 539.168,Z 1076.017,A -85,B 0,C 180,E1 11753.401,E2 11753.401} C_VEL
LIN {X 0,Y 526.134,Z 1131.409,A -85,B 0,C 180,E1 11761.165,E2 11761.165} C_VEL
LIN {X 0,Y 521.72,Z 1152.13,A -85,B 0,C 180,E1 11765.014,E2 11765.014} C_VEL
LIN {X 0,Y 511.474,Z 1168.285,A -85,B 0,C 180,E1 11768.331,E2 11768.331} C_VEL
LIN {X 0,Y 508.153,Z 1195.399,A -85,B 0,C 180,E1 11777.106,E2 11777.106} C_VEL
LIN {X 0,Y 507.293,Z 1206.844,A -85,B 0,C 180,E1 11784.037,E2 11784.037} C_VEL
LIN {X 0,Y 507.071,Z 1209.864,A -85,B 0,C 180,E1 11790.903,E2 11790.903} C_VEL
LIN {X 0,Y 507.207,Z 1203.738,A -85,B 0,C 180,E1 11798.445,E2 11798.445} C_VEL
LIN {X 0,Y 509.313,Z 1184.3,A -85,B 0,C 180,E1 11807.077,E2 11807.077} C_VEL
LIN {X 0,Y 515.166,Z 1149.279,A -85,B 0,C 180,E1 11815.955,E2 11815.955} C_VEL
LIN {X 0,Y 527.106,Z 1097.922,A -85,B 0,C 180,E1 11824.478,E2 11824.478} C_VEL
LIN {X 0,Y 541.746,Z 1041.43,A -85,B 0,C 180,E1 11830.77,E2 11830.77} C_VEL
LIN {X 0,Y 553.887,Z 976.386,A -85,B 0,C 180,E1 11835.295,E2 11835.295} C_VEL
LIN {X 0,Y 565.858,Z 892.062,A -85,B 0,C 180,E1 11838.903,E2 11838.903} C_VEL
LIN {X 0,Y 567.573,Z 865.412,A -85,B 0,C 180,E1 11839.834,E2 11839.834} C_VEL
LIN {X 0,Y 537.728,Z 810.596,A -85,B 0,C 180,E1 11845.588,E2 11845.588} C_VEL
LIN {X 0,Y 506.2,Z 762.06,A -85,B 0,C 180,E1 11853.226,E2 11853.226} C_VEL
LIN {X 0,Y 506.193,Z 762.06,A -85,B 0,C 180,E1 11863.404,E2 11863.404} C_VEL
LIN {X 0,Y 506.65,Z 762.06,A -85,B 0,C 180,E1 11872.204,E2 11872.204} C_VEL
LIN {X 0,Y 506.816,Z 762.06,A -85,B 0,C 180,E1 11880.807,E2 11880.807} C_VEL
LIN {X 0,Y 506.453,Z 762.06,A -85,B 0,C 180,E1 11889.433,E2 11889.433} C_VEL
LIN {X 0,Y 505.967,Z 762.06,A -85,B 0,C 180,E1 11899.013,E2 11899.013} C_VEL
LIN {X 0,Y 505.912,Z 762.06,A -85,B 0,C 180,E1 11907.679,E2 11907.679} C_VEL
LIN {X 0,Y 506.153,Z 764.16,A -85,B 0,C 180,E1 11910.642,E2 11910.642} C_VEL
LIN {X 0,Y 535.595,Z 811.586,A -85,B 0,C 180,E1 11917.27,E2 11917.27} C_VEL
LIN {X 0,Y 557.921,Z 867.154,A -85,B 0,C 180,E1 11922.123,E2 11922.123} C_VEL
LIN {X 0,Y 546.393,Z 947.559,A -85,B 0,C 180,E1 11925.905,E2 11925.905} C_VEL
LIN {X 0,Y 533.914,Z 1024.19,A -85,B 0,C 180,E1 11931.393,E2 11931.393} C_VEL
LIN {X 0,Y 523.151,Z 1079.786,A -85,B 0,C 180,E1 11937.497,E2 11937.497} C_VEL
LIN {X 0,Y 514.314,Z 1122.313,A -85,B 0,C 180,E1 11944.624,E2 11944.624} C_VEL
LIN {X 0,Y 509.136,Z 1156.144,A -85,B 0,C 180,E1 11953.506,E2 11953.506} C_VEL
LIN {X 0,Y 507.219,Z 1174.678,A -85,B 0,C 180,E1 11962.218,E2 11962.218} C_VEL
LIN {X 0,Y 506.793,Z 1179.896,A -85,B 0,C 180,E1 11969.097,E2 11969.097} C_VEL
LIN {X 0,Y 507.282,Z 1175.794,A -85,B 0,C 180,E1 11976.826,E2 11976.826} C_VEL
LIN {X 0,Y 508.784,Z 1158.691,A -85,B 0,C 180,E1 11985.522,E2 11985.522} C_VEL
LIN {X 0,Y 513.305,Z 1127.566,A -85,B 0,C 180,E1 11994.145,E2 11994.145} C_VEL
LIN {X 0,Y 521.611,Z 1087.065,A -85,B 0,C 180,E1 12001.386,E2 12001.386} C_VEL
LIN {X 0,Y 532.369,Z 1032.612,A -85,B 0,C 180,E1 12007.736,E2 12007.736} C_VEL
LIN {X 0,Y 543.77,Z 963.823,A -85,B 0,C 180,E1 12012.993,E2 12012.993} C_VEL
LIN {X 0,Y 556.039,Z 881.87,A -85,B 0,C 180,E1 12017.25,E2 12017.25} C_VEL
LIN {X 0,Y 557.74,Z 863.121,A -85,B 0,C 180,E1 12018.003,E2 12018.003} C_VEL
LIN {X 0,Y 538.63,Z 819.739,A -85,B 0,C 180,E1 12021.958,E2 12021.958} C_VEL
LIN {X 0,Y 516.059,Z 840.682,A -85,B 0,C 180,E1 12024.184,E2 12024.184} C_VEL
LIN {X 0,Y 513.756,Z 866.687,A -85,B 0,C 180,E1 12025.341,E2 12025.341} C_VEL
LIN {X 0,Y 513.165,Z 995.357,A -85,B 0,C 180,E1 12027.571,E2 12027.571} C_VEL
LIN {X 0,Y 512.026,Z 1035.177,A -85,B 0,C 180,E1 12029.95,E2 12029.95} C_VEL
LIN {X 0,Y 510.458,Z 1065.354,A -85,B 0,C 180,E1 12033.647,E2 12033.647} C_VEL
LIN {X 0,Y 509.471,Z 1082.256,A -85,B 0,C 180,E1 12038.199,E2 12038.199} C_VEL
LIN {X 0,Y 509.541,Z 1084.225,A -85,B 0,C 180,E1 12042.852,E2 12042.852} C_VEL
LIN {X 0,Y 510.649,Z 1071.576,A -85,B 0,C 180,E1 12047.389,E2 12047.389} C_VEL
LIN {X 0,Y 511.752,Z 1045.464,A -85,B 0,C 180,E1 12051.203,E2 12051.203} C_VEL
LIN {X 0,Y 512.968,Z 1007.994,A -85,B 0,C 180,E1 12053.852,E2 12053.852} C_VEL
LIN {X 0,Y 513.013,Z 957.355,A -85,B 0,C 180,E1 12055.119,E2 12055.119} C_VEL
LIN {X 0,Y 514.888,Z 858.415,A -85,B 0,C 180,E1 12056.882,E2 12056.882} C_VEL
LIN {X 0,Y 514.081,Z 794.206,A -85,B 0,C 180,E1 12059.733,E2 12059.733} C_VEL
LIN {X 0,Y 506.575,Z 762.06,A -85,B 0,C 180,E1 12061.499,E2 12061.499} C_VEL
LIN {X 0,Y 506.312,Z 762.06,A -85,B 0,C 180,E1 12069.538,E2 12069.538} C_VEL
LIN {X 0,Y 505.976,Z 762.06,A -85,B 0,C 180,E1 12079.294,E2 12079.294} C_VEL
LIN {X 0,Y 506.021,Z 763.828,A -85,B 0,C 180,E1 12087.206,E2 12087.206} C_VEL
LIN {X 0,Y 542.107,Z 818.179,A -85,B 0,C 180,E1 12095.315,E2 12095.315} C_VEL
LIN {X 0,Y 568.765,Z 868.355,A -85,B 0,C 180,E1 12100.412,E2 12100.412} C_VEL
LIN {X 0,Y 557.575,Z 953.773,A -85,B 0,C 180,E1 12103.553,E2 12103.553} C_VEL
LIN {X 0,Y 545.403,Z 1024.122,A -85,B 0,C 180,E1 12107.813,E2 12107.813} C_VEL
LIN {X 0,Y 532.712,Z 1077.055,A -85,B 0,C 180,E1 12112.884,E2 12112.884} C_VEL
LIN {X 0,Y 518.805,Z 1131.706,A -85,B 0,C 180,E1 12120.733,E2 12120.733} C_VEL
LIN {X 0,Y 511.474,Z 1168.285,A -85,B 0,C 180,E1 12128.331,E2 12128.331} C_VEL
LIN {X 0,Y 501.524,Z 1182.015,A -85,B 0,C 180,E1 12131.879,E2 12131.879} C_VEL
LIN {X 0,Y 499.35,Z 1200.717,A -85,B 0,C 180,E1 12139.542,E2 12139.542} C_VEL
LIN {X 0,Y 499.125,Z 1209.387,A -85,B 0,C 180,E1 12147.433,E2 12147.433} C_VEL
LIN {X 0,Y 499.196,Z 1208.305,A -85,B 0,C 180,E1 12154.404,E2 12154.404} C_VEL
LIN {X 0,Y 499.854,Z 1197.128,A -85,B 0,C 180,E1 12162.315,E2 12162.315} C_VEL
LIN {X 0,Y 502.67,Z 1173.123,A -85,B 0,C 180,E1 12170.745,E2 12170.745} C_VEL
LIN {X 0,Y 510.957,Z 1133.895,A -85,B 0,C 180,E1 12179.391,E2 12179.391} C_VEL
LIN {X 0,Y 525.546,Z 1080.822,A -85,B 0,C 180,E1 12187.366,E2 12187.366} C_VEL
LIN {X 0,Y 538.179,Z 1030.416,A -85,B 0,C 180,E1 12192.303,E2 12192.303} C_VEL
LIN {X 0,Y 550.935,Z 958.632,A -85,B 0,C 180,E1 12196.771,E2 12196.771} C_VEL
LIN {X 0,Y 561.596,Z 868.991,A -85,B 0,C 180,E1 12200.341,E2 12200.341} C_VEL
LIN {X 0,Y 533.381,Z 816.167,A -85,B 0,C 180,E1 12206.007,E2 12206.007} C_VEL
LIN {X 0,Y 501.472,Z 768.516,A -85,B 0,C 180,E1 12213.572,E2 12213.572} C_VEL
LIN {X 0,Y 498.138,Z 762.06,A -85,B 0,C 180,E1 12214.703,E2 12214.703} C_VEL
LIN {X 0,Y 498.17,Z 762.06,A -85,B 0,C 180,E1 12224.943,E2 12224.943} C_VEL
LIN {X 0,Y 498.478,Z 762.06,A -85,B 0,C 180,E1 12233.833,E2 12233.833} C_VEL
LIN {X 0,Y 498.809,Z 762.06,A -85,B 0,C 180,E1 12240.82,E2 12240.82} C_VEL
LIN {X 0,Y 498.417,Z 762.06,A -85,B 0,C 180,E1 12249.586,E2 12249.586} C_VEL
LIN {X 0,Y 497.967,Z 762.06,A -85,B 0,C 180,E1 12258.604,E2 12258.604} C_VEL
LIN {X 0,Y 497.883,Z 762.06,A -85,B 0,C 180,E1 12268.129,E2 12268.129} C_VEL
LIN {X 0,Y 498.389,Z 764.906,A -85,B 0,C 180,E1 12269.115,E2 12269.115} C_VEL
LIN {X 0,Y 525.983,Z 807.885,A -85,B 0,C 180,E1 12275.809,E2 12275.809} C_VEL
LIN {X 0,Y 541.399,Z 842.321,A -85,B 0,C 180,E1 12279.175,E2 12279.175} C_VEL
LIN {X 0,Y 551.653,Z 871.14,A -85,B 0,C 180,E1 12281.673,E2 12281.673} C_VEL
LIN {X 0,Y 539.595,Z 950.518,A -85,B 0,C 180,E1 12285.538,E2 12285.538} C_VEL
LIN {X 0,Y 525.093,Z 1031.77,A -85,B 0,C 180,E1 12291.738,E2 12291.738} C_VEL
LIN {X 0,Y 514.646,Z 1085.154,A -85,B 0,C 180,E1 12297.895,E2 12297.895} C_VEL
LIN {X 0,Y 506.135,Z 1126.452,A -85,B 0,C 180,E1 12305.134,E2 12305.134} C_VEL
LIN {X 0,Y 500.871,Z 1158.675,A -85,B 0,C 180,E1 12314.13,E2 12314.13} C_VEL
LIN {X 0,Y 499.093,Z 1175.789,A -85,B 0,C 180,E1 12322.969,E2 12322.969} C_VEL
LIN {X 0,Y 499.111,Z 1179.893,A -85,B 0,C 180,E1 12330.825,E2 12330.825} C_VEL
LIN {X 0,Y 499.446,Z 1172.276,A -85,B 0,C 180,E1 12339.455,E2 12339.455} C_VEL
LIN {X 0,Y 501.117,Z 1153.223,A -85,B 0,C 180,E1 12347.664,E2 12347.664} C_VEL
LIN {X 0,Y 506.655,Z 1121.323,A -85,B 0,C 180,E1 12355.902,E2 12355.902} C_VEL
LIN {X 0,Y 515.645,Z 1078.609,A -85,B 0,C 180,E1 12362.929,E2 12362.929} C_VEL
LIN {X 0,Y 526.562,Z 1023.95,A -85,B 0,C 180,E1 12368.886,E2 12368.886} C_VEL
LIN {X 0,Y 541.117,Z 942.704,A -85,B 0,C 180,E1 12374.813,E2 12374.813} C_VEL
LIN {X 0,Y 551.323,Z 866.172,A -85,B 0,C 180,E1 12378.527,E2 12378.527} C_VEL
LIN {X 0,Y 535.855,Z 830.335,A -85,B 0,C 180,E1 12381.91,E2 12381.91} C_VEL
LIN {X 0,Y 512.249,Z 854.471,A -85,B 0,C 180,E1 12384.058,E2 12384.058} C_VEL
LIN {X 0,Y 506.187,Z 859.879,A -85,B 0,C 180,E1 12384.944,E2 12384.944} C_VEL
LIN {X 0,Y 505.384,Z 996.179,A -85,B 0,C 180,E1 12387.385,E2 12387.385} C_VEL
LIN {X 0,Y 504.22,Z 1035.665,A -85,B 0,C 180,E1 12389.761,E2 12389.761} C_VEL
LIN {X 0,Y 502.595,Z 1065.845,A -85,B 0,C 180,E1 12393.46,E2 12393.46} C_VEL
LIN {X 0,Y 501.547,Z 1082.612,A -85,B 0,C 180,E1 12397.836,E2 12397.836} C_VEL
